// ---- VISUs/Estufa2.TcVIS
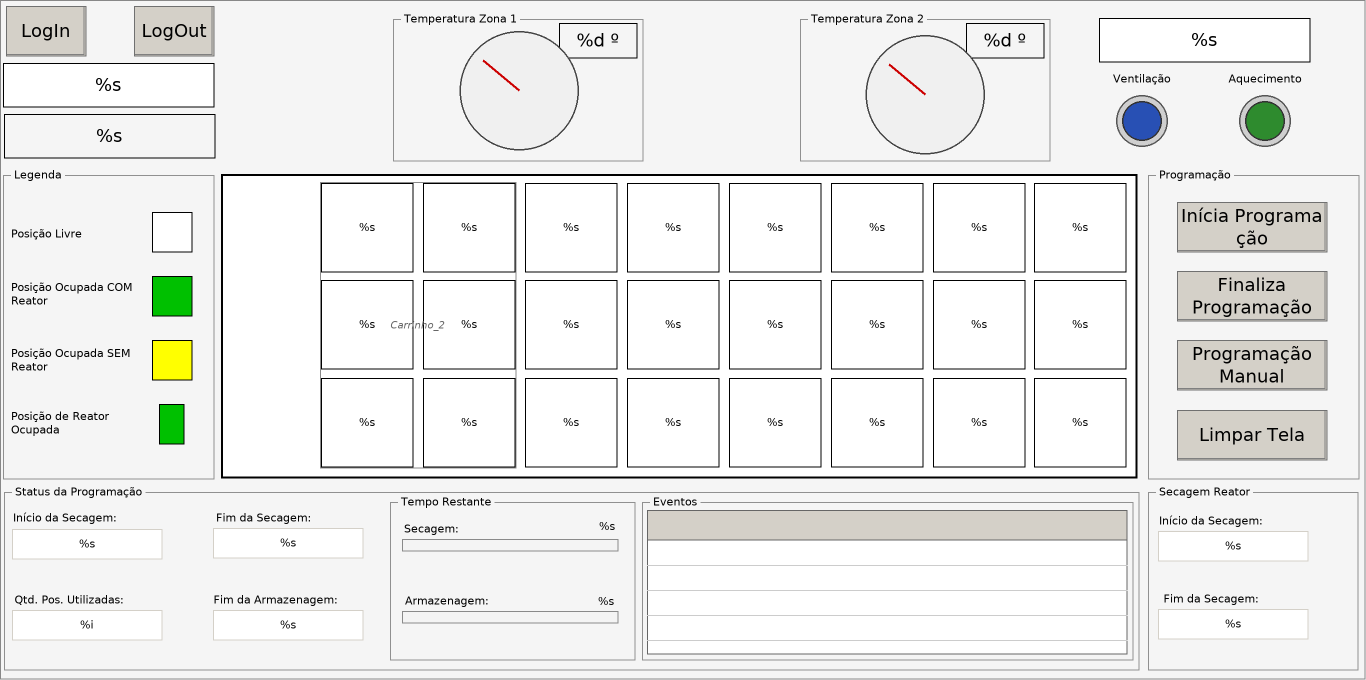
VISUALIZATION Estufa2  // 1366x680
    GroupBox (1148,484 210x186), "Secagem Reator", invisible if: GVL_P.bCarrinhoReator2
        Label (10,100 106x30), "Fim da Secagem:"
        Textfield (10,125 150x30), "%s", text variable: GVL_P.arrStatusEstufas[1].statusFimSecagem
    GroupBox (3,167 211x312), "Legenda"
        RoundedRectangle (149,173 40x40)
        RoundedRectangle (149,45 40x40)
        RoundedRectangle (156,237 25x40)
    GroupBox (800,11 250x150), "Temperatura Zona 2"
        Rectangle (166,12 78x35), "%d º", text variable: GVL.zona2atual_020
    GroupBox (393,11 250x150), "Temperatura Zona 1"
        Rectangle (166,12 78x35), "%d º", text variable: GVL.zona1atual_020
    GroupBox (4,484 1135x186), "Status da Programação"
        Label (209,19 101x30), "Fim da Secagem:"
        Label (209,101 125x30), "Fim da Armazenagem:"
        Label (8,101 114x30), "Qtd. Pos. Utilizadas:"
        GroupBox (638,10 491x166), "Eventos"
            Table (5,16 480x144), data array: GVL_P.arrLogEstufa20
                p3854506369: GVL_P.arrLogEstufa20[INDEX]
            InvisibleInput (7,16 431x142)
                OnMouseClick: OpenDialog Dialog=addComment, OpenModal=True, OpenCentered=True
        Label (8,19 106x30), "Início da Secagem:"
        Textfield (8,126 150x30), "%i", text variable: GVL.totalPos[1]
        Textfield (209,44 150x30), "%s", text variable: GVL_P.arrStatusEstufas[1].statusFimSecagem
        Textfield (209,126 150x30), "%s", text variable: GVL_P.arrStatusEstufas[1].statusFimArmazenagem
        GroupBox (386,10 245x166), "Tempo Restante"
            Progressbar (12,117 216x12), variable: MAIN.bardintArm20
            Rectangle (131,99 96x17), "%s", text variable: mid(str:=time_to_string(GVL.endArm20), LEN:= 20, POS:= 3)
            Progressbar (12,45 216x12), variable: MAIN.bardintSec20
        Label (398,30 59x30), "Secagem:"
    Rectangle (221,174 916x304)
    Meter180 (399,31 240x119), value: GVL.zona1atual_020, style: Meter-Meter180-Gray, scale format: %.1f, scale 20..160
        p518627256: ºC
    GroupBox (1148,167 211x312), "Programação"
        Button (29,35 150x50), "Inícia Programação", input disabled if: GVL_P.arrStatusEstufas[GVL.actEst].start
            OnMouseClick: OpenDialog Dialog=IniciaProg_2, OpenModal=True, OpenCentered=True
            OnMouseClick: execute { iniciaProgramacaoEstufa(); }
        Button (29,104 150x50), "Finaliza Programação"
            OnMouseClick: OpenDialog Dialog=FinalizaProg, Parameters={bReator: , iOFnumber: , iSrlNumber: }, OpenModal=True, OpenCentered=True
        Button (29,173 150x50), "Programação Manual", input disabled if: GVL_P.arrStatusEstufas[GVL.actEst].start
            OnMouseClick: OpenDialog Dialog=TimeCustom_2, OpenModal=True, OpenCentered=True
            OnMouseClick: execute { iniciaProgramacaoEstufa(); }
    Textfield (12,529 150x30), "%s", text variable: GVL_P.arrStatusEstufas[1].statusInicioSecagem
    Label (402,586 90x30), "Armazenagem:"
    Meter180 (805,35 240x119), value: GVL.zona2atual_020, style: Meter-Meter180-Gray, scale format: %.1f, scale 20..160
        p518627256: ºC
    RoundedRectangle (152,276 40x40)
    Label (8,278 132x32), "Posição Ocupada COM Reator"
    Label (8,344 128x32), "Posição Ocupada SEM Reator"
    Label (8,218 84x32), "Posição Livre"
    Label (8,407 128x32), "Posição de Reator Ocupada"
    Lamp1 (1112,91 60x60), variable: GVL.ventilacao_Ligada_020, style: Lamp-Lamp1-Blue
    Lamp1 (1235,91 60x60), variable: GVL.aquecimento_Ligado_020, style: Lamp-Lamp1-Green
    Label (1108,64 68x30), "Ventilação"
    Label (1227,64 76x30), "Aquecimento"
    Textfield (1158,531 150x30), "%s", text variable: GVL_P.arrStatusEstufas[1].inicioReator, invisible if: GVL_P.bCarrinhoReator2
    Label (1158,506 106x30), "Início da Secagem:", invisible if: GVL_P.bCarrinhoReator2
    Rectangle (1099,18 211x44), "%s", text variable: GVL_P.etapa_process[GVL.actEst]
    Rectangle (522,518 96x17), "%s", text variable: mid(str:=time_to_string(GVL.endSeca20), LEN:= 20, POS:= 3)
    Rectangle (1034,183 92x89), "%s", text variable: GVL_P.aPositionsE020[1].text, colour variable: GVL_P.aPositionsE020[1].color
        OnMouseUp: OpenDialog Dialog=ConfigPosicao_2, Parameters={bReator: , iOFnumber: , iSrlNumber: }, OpenModal=True, OpenCentered=True
        OnMouseUp: execute {
            gvl.actPos:=1;
            //selectPos021();
        }
    Rectangle (1034,280 92x89), "%s", text variable: GVL_P.aPositionsE020[2].text, colour variable: GVL_P.aPositionsE020[2].color
        OnMouseUp: OpenDialog Dialog=ConfigPosicao_2, Parameters={bReator: , iOFnumber: , iSrlNumber: }, OpenModal=True, OpenCentered=True
        OnMouseUp: execute {
            gvl.actPos:= 2;
            //selectPos021();
        }
    Rectangle (1034,378 92x89), "%s", text variable: GVL_P.aPositionsE020[3].text, colour variable: GVL_P.aPositionsE020[3].color
        OnMouseUp: OpenDialog Dialog=ConfigPosicao_2, Parameters={bReator: , iOFnumber: , iSrlNumber: }, OpenModal=True, OpenCentered=True
        OnMouseUp: execute {
            gvl.actPos:= 3;
            //selectPos021();
        }
    Rectangle (933,183 92x89), "%s", text variable: GVL_P.aPositionsE020[4].text, colour variable: GVL_P.aPositionsE020[4].color
        OnMouseUp: OpenDialog Dialog=ConfigPosicao_2, Parameters={bReator: , iOFnumber: , iSrlNumber: }, OpenModal=True, OpenCentered=True
        OnMouseUp: execute {
            gvl.actPos:= 4;
            //selectPos021();
        }
    Rectangle (933,280 92x89), "%s", text variable: GVL_P.aPositionsE020[5].text, colour variable: GVL_p.aPositionsE020[5].color
        OnMouseUp: OpenDialog Dialog=ConfigPosicao_2, Parameters={bReator: , iOFnumber: , iSrlNumber: }, OpenModal=True, OpenCentered=True
        OnMouseUp: execute {
            gvl.actPos:= 5;
            //selectPos021();
        }
    Rectangle (933,378 92x89), "%s", text variable: GVL_P.aPositionsE020[6].text, colour variable: GVL_P.aPositionsE020[6].color
        OnMouseUp: OpenDialog Dialog=ConfigPosicao_2, Parameters={bReator: , iOFnumber: , iSrlNumber: }, OpenModal=True, OpenCentered=True
        OnMouseUp: execute {
            gvl.actPos:= 6;
            //selectPos021();
        }
    Rectangle (831,183 92x89), "%s", text variable: GVL_P.aPositionsE020[7].text, colour variable: GVL_P.aPositionsE020[7].color
        OnMouseUp: OpenDialog Dialog=ConfigPosicao_2, Parameters={bReator: , iOFnumber: , iSrlNumber: }, OpenModal=True, OpenCentered=True
        OnMouseUp: execute {
            gvl.actPos:= 7;
            //selectPos021();
        }
    Rectangle (831,280 92x89), "%s", text variable: GVL_P.aPositionsE020[8].text, colour variable: GVL_P.aPositionsE020[8].color
        OnMouseUp: OpenDialog Dialog=ConfigPosicao_2, Parameters={bReator: , iOFnumber: , iSrlNumber: }, OpenModal=True, OpenCentered=True
        OnMouseUp: execute {
            gvl.actPos:= 8;
            //selectPos021();
        }
    Rectangle (831,378 92x89), "%s", text variable: GVL_P.aPositionsE020[9].text, colour variable: GVL_P.aPositionsE020[9].color
        OnMouseUp: OpenDialog Dialog=ConfigPosicao_2, Parameters={bReator: , iOFnumber: , iSrlNumber: }, OpenModal=True, OpenCentered=True
        OnMouseUp: execute {
            gvl.actPos:= 9;
            //selectPos021();
        }
    Rectangle (729,183 92x89), "%s", text variable: GVL_P.aPositionsE020[10].text, colour variable: GVL_P.aPositionsE020[10].color
        OnMouseUp: OpenDialog Dialog=ConfigPosicao_2, Parameters={bReator: , iOFnumber: , iSrlNumber: }, OpenModal=True, OpenCentered=True
        OnMouseUp: execute {
            gvl.actPos:= 10;
            //selectPos021();
        }
    Rectangle (729,280 92x89), "%s", text variable: GVL_P.aPositionsE020[11].text, colour variable: GVL_P.aPositionsE020[11].color
        OnMouseUp: OpenDialog Dialog=ConfigPosicao_2, Parameters={bReator: , iOFnumber: , iSrlNumber: }, OpenModal=True, OpenCentered=True
        OnMouseUp: execute {
            gvl.actPos:= 11;
            //selectPos021();
        }
    Rectangle (729,378 92x89), "%s", text variable: GVL_P.aPositionsE020[12].text, colour variable: GVL_P.aPositionsE020[12].color
        OnMouseUp: OpenDialog Dialog=ConfigPosicao_2, Parameters={bReator: , iOFnumber: , iSrlNumber: }, OpenModal=True, OpenCentered=True
        OnMouseUp: execute {
            gvl.actPos:= 12;
            //selectPos021();
        }
    Rectangle (627,183 92x89), "%s", text variable: GVL_P.aPositionsE020[13].text, colour variable: GVL_P.aPositionsE020[13].color
        OnMouseUp: OpenDialog Dialog=ConfigPosicao_2, Parameters={bReator: , iOFnumber: , iSrlNumber: }, OpenModal=True, OpenCentered=True
        OnMouseUp: execute {
            gvl.actPos:= 13;
            //selectPos021();
        }
    Rectangle (627,280 92x89), "%s", text variable: GVL_P.aPositionsE020[14].text, colour variable: GVL_P.aPositionsE020[14].color
        OnMouseUp: OpenDialog Dialog=ConfigPosicao_2, Parameters={bReator: , iOFnumber: , iSrlNumber: }, OpenModal=True, OpenCentered=True
        OnMouseUp: execute {
            gvl.actPos:= 14;
            //selectPos021();
        }
    Rectangle (627,378 92x89), "%s", text variable: GVL_P.aPositionsE020[15].text, colour variable: GVL_P.aPositionsE020[15].color
        OnMouseUp: OpenDialog Dialog=ConfigPosicao_2, Parameters={bReator: , iOFnumber: , iSrlNumber: }, OpenModal=True, OpenCentered=True
        OnMouseUp: execute {
            gvl.actPos:= 15;
            //selectPos021();
        }
    Rectangle (525,183 92x89), "%s", text variable: GVL_P.aPositionsE020[16].text, colour variable: GVL_P.aPositionsE020[16].color
        OnMouseUp: OpenDialog Dialog=ConfigPosicao_2, Parameters={bReator: , iOFnumber: , iSrlNumber: }, OpenModal=True, OpenCentered=True
        OnMouseUp: execute {
            gvl.actPos:= 16;
            //selectPos021();
        }
    Rectangle (525,280 92x89), "%s", text variable: GVL_P.aPositionsE020[17].text, colour variable: GVL_P.aPositionsE020[17].color
        OnMouseUp: OpenDialog Dialog=ConfigPosicao_2, Parameters={bReator: , iOFnumber: , iSrlNumber: }, OpenModal=True, OpenCentered=True
        OnMouseUp: execute {
            gvl.actPos:= 17;
            //selectPos021();
        }
    Rectangle (525,378 92x89), "%s", text variable: GVL_P.aPositionsE020[18].text, colour variable: GVL_P.aPositionsE020[18].color
        OnMouseUp: OpenDialog Dialog=ConfigPosicao_2, Parameters={bReator: , iOFnumber: , iSrlNumber: }, OpenModal=True, OpenCentered=True
        OnMouseUp: execute {
            gvl.actPos:= 18;
            //selectPos021();
        }
    Rectangle (423,183 92x89), "%s", text variable: GVL_P.aPositionsE020[19].text, colour variable: GVL_P.aPositionsE020[19].color
        OnMouseUp: OpenDialog Dialog=ConfigPosicao_2, Parameters={bReator: , iOFnumber: , iSrlNumber: }, OpenModal=True, OpenCentered=True
        OnMouseUp: execute {
            gvl.actPos:= 19;
            //selectPos021();
        }
    Rectangle (423,280 92x89), "%s", text variable: GVL_P.aPositionsE020[20].text, colour variable: GVL_P.aPositionsE020[20].color
        OnMouseUp: OpenDialog Dialog=ConfigPosicao_2, Parameters={bReator: , iOFnumber: , iSrlNumber: }, OpenModal=True, OpenCentered=True
        OnMouseUp: execute {
            gvl.actPos:= 20;
            //selectPos021();
        }
    Rectangle (423,378 92x89), "%s", text variable: GVL_P.aPositionsE020[21].text, colour variable: GVL_P.aPositionsE020[21].color
        OnMouseUp: OpenDialog Dialog=ConfigPosicao_2, Parameters={bReator: , iOFnumber: , iSrlNumber: }, OpenModal=True, OpenCentered=True
        OnMouseUp: execute {
            gvl.actPos:= 21;
            //selectPos021();
        }
    Rectangle (321,183 92x89), "%s", text variable: GVL_P.aPositionsE020[22].text, colour variable: GVL_P.aPositionsE020[22].color
        OnMouseUp: OpenDialog Dialog=ConfigPosicao_2, Parameters={bReator: , iOFnumber: , iSrlNumber: }, OpenModal=True, OpenCentered=True
        OnMouseUp: execute {
            gvl.actPos:= 22;
            //selectPos021();
        }
    Rectangle (321,280 92x89), "%s", text variable: GVL_P.aPositionsE020[23].text, colour variable: GVL_P.aPositionsE020[23].color
        OnMouseUp: OpenDialog Dialog=ConfigPosicao_2, Parameters={bReator: , iOFnumber: , iSrlNumber: }, OpenModal=True, OpenCentered=True
        OnMouseUp: execute {
            gvl.actPos:= 23;
            //selectPos021();
        }
    Rectangle (321,378 92x89), "%s", text variable: GVL_P.aPositionsE020[24].text, colour variable: GVL_P.aPositionsE020[24].color
        OnMouseUp: OpenDialog Dialog=ConfigPosicao_2, Parameters={bReator: , iOFnumber: , iSrlNumber: }, OpenModal=True, OpenCentered=True
        OnMouseUp: execute {
            gvl.actPos:= 24;
            //selectPos021();
        }
    Frame (320,182 196x286), invisible if: GVL_P.bCarrinhoReator2
        shows Carrinho_2()
    Button (1177,410 150x50), "Limpar Tela"
        OnMouseClick: execute {
            FOR gvl.i:=1 TO 24 BY 1 DO
            gvl_p.aPositionsE020[gvl.i].numOF:='';
            gvl_p.aPositionsE020[gvl.i].lote:='';
            gvl_p.aPositionsE020[gvl.i].class:=0;
            gvl_p.aPositionsE020[gvl.i].pot:=0;
            gvl_p.aPositionsE020[gvl.i].cor:=0;
            gvl_p.aPositionsE020[gvl.i].text:='';
            gvl_p.aPositionsE020[gvl.i].reator:=true;
            END_FOR
            FOR gvl.i:=1 TO 18 BY 1 DO
            gvl_p.corPosReator2[gvl.i].cor:=0;
            END_FOR
            gravarConfigPosicao.bReator[1]:= FALSE;
            ///// GERADOR DE LOG -------------------------------------------------------------
            gvl.envialog:= 'Todas as posições foram limpas. ESTUFA 20';
            gvl.logRegister20:= gvl.envialog;
            gvl.sCmdInsertLog:= 'INSERT INTO [dbo].[LogGeneral] ([HistoricalTime],[Description])VALUES($'$',$'$')';
            gvl.sCmdInsertLog:= insert(gvl.sCmdInsertLog,gvl.logRegister20,74);
            gvl.sCmdInsertLog:= insert(gvl.sCmdInsertLog,gvl.sSystemDateTime,71);
            gvl.bInsertLog:= TRUE;
        }
    Rectangle (3,63 211x44), "%s", text variable: MAIN.sDB_Operador
    Rectangle (4,114 211x44), "%s", text variable: GVL.sSystemTime
    Button (6,6 80x50), "LogIn"
        OnMouseClick: VisuUserMgmt Type=Login
    Button (134,6 80x50), "LogOut"
        OnMouseClick: VisuUserMgmt Type=Logout
END_VISUALIZATION

// ---- VISUs/Estufa3.TcVIS
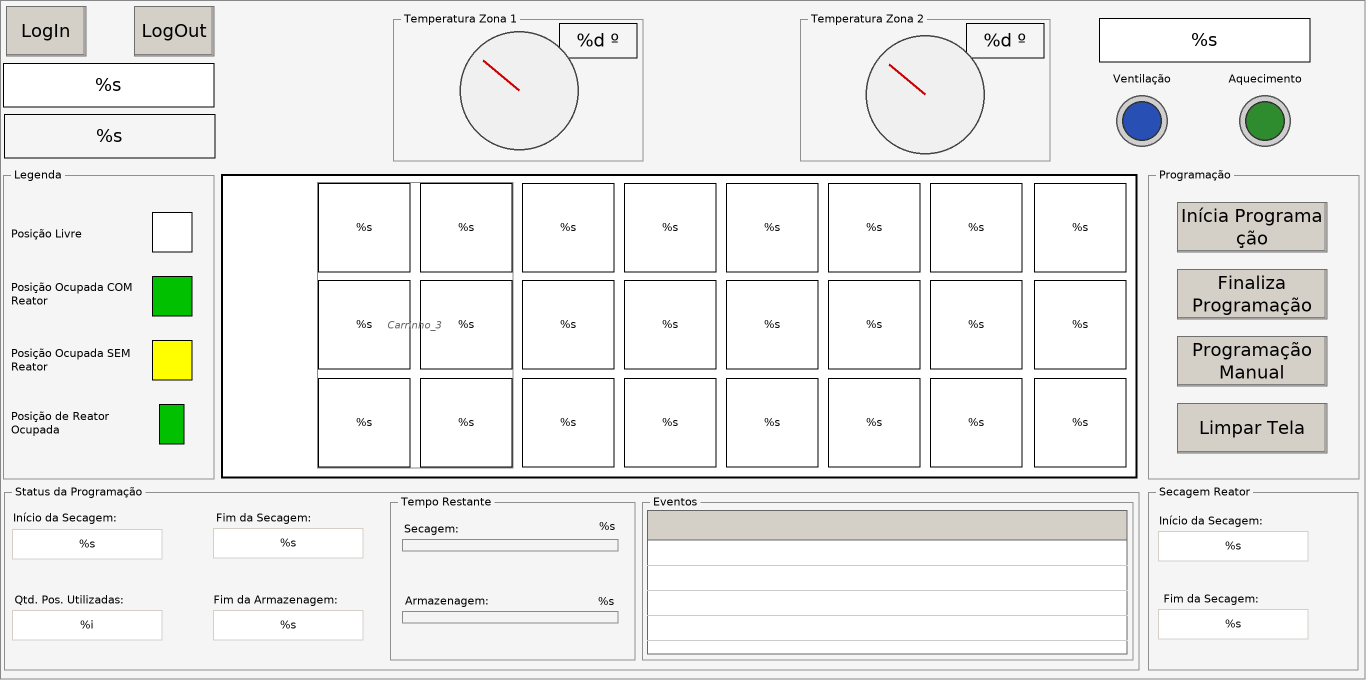
VISUALIZATION Estufa3  // 1366x680
    GroupBox (1148,484 210x186), "Secagem Reator", invisible if: GVL_P.bCarrinhoReator3
        Label (10,100 106x30), "Fim da Secagem:"
        Textfield (10,125 150x30), "%s", text variable: GVL_P.arrStatusEstufas[2].statusFimSecagem
    GroupBox (3,167 211x312), "Legenda"
        RoundedRectangle (149,173 40x40)
        RoundedRectangle (149,45 40x40)
        RoundedRectangle (156,237 25x40)
    GroupBox (800,11 250x150), "Temperatura Zona 2"
        Rectangle (166,12 78x35), "%d º", text variable: GVL.zona2atual_021
    GroupBox (393,11 250x150), "Temperatura Zona 1"
        Rectangle (166,12 78x35), "%d º", text variable: GVL.zona1atual_021
    GroupBox (4,484 1135x186), "Status da Programação"
        Label (209,19 101x30), "Fim da Secagem:"
        Label (209,101 125x30), "Fim da Armazenagem:"
        Label (8,101 114x30), "Qtd. Pos. Utilizadas:"
        GroupBox (638,10 491x166), "Eventos"
            Table (5,16 480x144), data array: GVL_P.arrLogEstufa21
                p3854506369: GVL_P.arrLogEstufa21[INDEX]
            InvisibleInput (7,16 431x142)
                OnMouseClick: OpenDialog Dialog=addComment, OpenModal=True, OpenCentered=True
        Label (8,19 106x30), "Início da Secagem:"
        Textfield (8,126 150x30), "%i", text variable: GVL.totalPos[2]
        Textfield (209,44 150x30), "%s", text variable: GVL_P.arrStatusEstufas[2].statusFimSecagem
        Textfield (209,126 150x30), "%s", text variable: GVL_P.arrStatusEstufas[2].statusFimArmazenagem
        GroupBox (386,10 245x166), "Tempo Restante"
            Progressbar (12,117 216x12), variable: MAIN.bardintArm21
            Rectangle (131,99 96x17), "%s", text variable: mid(str:=time_to_string(GVL.endArm21), LEN:= 20, POS:= 3)
            Progressbar (12,45 216x12), variable: MAIN.bardintSec21
        Label (398,30 59x30), "Secagem:"
    Rectangle (221,174 916x304)
    Rectangle (1034,183 92x89), "%s", text variable: GVL_P.aPositionsE021[1].text, colour variable: GVL_P.aPositionsE021[1].color
        OnMouseUp: OpenDialog Dialog=ConfigPosicao_3, Parameters={bReator: , iOFnumber: , iSrlNumber: }, OpenModal=True, OpenCentered=True
        OnMouseUp: execute {
            gvl.actPos:=1;
            //selectPos021();
        }
    Rectangle (1034,280 92x89), "%s", text variable: GVL_P.aPositionsE021[2].text, colour variable: GVL_P.aPositionsE021[2].color
        OnMouseUp: OpenDialog Dialog=ConfigPosicao_3, Parameters={bReator: , iOFnumber: , iSrlNumber: }, OpenModal=True, OpenCentered=True
        OnMouseUp: execute {
            gvl.actPos:= 2;
            //selectPos021();
        }
    Rectangle (1034,378 92x89), "%s", text variable: GVL_P.aPositionsE021[3].text, colour variable: GVL_P.aPositionsE021[3].color
        OnMouseUp: OpenDialog Dialog=ConfigPosicao_3, Parameters={bReator: , iOFnumber: , iSrlNumber: }, OpenModal=True, OpenCentered=True
        OnMouseUp: execute {
            gvl.actPos:= 3;
            //selectPos021();
        }
    Rectangle (930,183 92x89), "%s", text variable: GVL_P.aPositionsE021[4].text, colour variable: GVL_P.aPositionsE021[4].color
        OnMouseUp: OpenDialog Dialog=ConfigPosicao_3, Parameters={bReator: , iOFnumber: , iSrlNumber: }, OpenModal=True, OpenCentered=True
        OnMouseUp: execute {
            gvl.actPos:= 4;
            //selectPos021();
        }
    Rectangle (930,280 92x89), "%s", text variable: GVL_P.aPositionsE021[5].text, colour variable: GVL_p.aPositionsE021[5].color
        OnMouseUp: OpenDialog Dialog=ConfigPosicao_3, Parameters={bReator: , iOFnumber: , iSrlNumber: }, OpenModal=True, OpenCentered=True
        OnMouseUp: execute {
            gvl.actPos:= 5;
            //selectPos021();
        }
    Rectangle (930,378 92x89), "%s", text variable: GVL_P.aPositionsE021[6].text, colour variable: GVL_P.aPositionsE021[6].color
        OnMouseUp: OpenDialog Dialog=ConfigPosicao_3, Parameters={bReator: , iOFnumber: , iSrlNumber: }, OpenModal=True, OpenCentered=True
        OnMouseUp: execute {
            gvl.actPos:= 6;
            //selectPos021();
        }
    Rectangle (828,183 92x89), "%s", text variable: GVL_P.aPositionsE021[7].text, colour variable: GVL_P.aPositionsE021[7].color
        OnMouseUp: OpenDialog Dialog=ConfigPosicao_3, Parameters={bReator: , iOFnumber: , iSrlNumber: }, OpenModal=True, OpenCentered=True
        OnMouseUp: execute {
            gvl.actPos:= 7;
            //selectPos021();
        }
    Rectangle (828,280 92x89), "%s", text variable: GVL_P.aPositionsE021[8].text, colour variable: GVL_P.aPositionsE021[8].color
        OnMouseUp: OpenDialog Dialog=ConfigPosicao_3, Parameters={bReator: , iOFnumber: , iSrlNumber: }, OpenModal=True, OpenCentered=True
        OnMouseUp: execute {
            gvl.actPos:= 8;
            //selectPos021();
        }
    Rectangle (828,378 92x89), "%s", text variable: GVL_P.aPositionsE021[9].text, colour variable: GVL_P.aPositionsE021[9].color
        OnMouseUp: OpenDialog Dialog=ConfigPosicao_3, Parameters={bReator: , iOFnumber: , iSrlNumber: }, OpenModal=True, OpenCentered=True
        OnMouseUp: execute {
            gvl.actPos:= 9;
            //selectPos021();
        }
    Rectangle (726,183 92x89), "%s", text variable: GVL_P.aPositionsE021[10].text, colour variable: GVL_P.aPositionsE021[10].color
        OnMouseUp: OpenDialog Dialog=ConfigPosicao_3, Parameters={bReator: , iOFnumber: , iSrlNumber: }, OpenModal=True, OpenCentered=True
        OnMouseUp: execute {
            gvl.actPos:= 10;
            //selectPos021();
        }
    Rectangle (726,280 92x89), "%s", text variable: GVL_P.aPositionsE021[11].text, colour variable: GVL_P.aPositionsE021[11].color
        OnMouseUp: OpenDialog Dialog=ConfigPosicao_3, Parameters={bReator: , iOFnumber: , iSrlNumber: }, OpenModal=True, OpenCentered=True
        OnMouseUp: execute {
            gvl.actPos:= 11;
            //selectPos021();
        }
    Rectangle (726,378 92x89), "%s", text variable: GVL_P.aPositionsE021[12].text, colour variable: GVL_P.aPositionsE021[12].color
        OnMouseUp: OpenDialog Dialog=ConfigPosicao_3, Parameters={bReator: , iOFnumber: , iSrlNumber: }, OpenModal=True, OpenCentered=True
        OnMouseUp: execute {
            gvl.actPos:= 12;
            //selectPos021();
        }
    Rectangle (624,183 92x89), "%s", text variable: GVL_P.aPositionsE021[13].text, colour variable: GVL_P.aPositionsE021[13].color
        OnMouseUp: OpenDialog Dialog=ConfigPosicao_3, Parameters={bReator: , iOFnumber: , iSrlNumber: }, OpenModal=True, OpenCentered=True
        OnMouseUp: execute {
            gvl.actPos:= 13;
            //selectPos021();
        }
    Rectangle (624,280 92x89), "%s", text variable: GVL_P.aPositionsE021[14].text, colour variable: GVL_P.aPositionsE021[14].color
        OnMouseUp: OpenDialog Dialog=ConfigPosicao_3, Parameters={bReator: , iOFnumber: , iSrlNumber: }, OpenModal=True, OpenCentered=True
        OnMouseUp: execute {
            gvl.actPos:= 14;
            //selectPos021();
        }
    Rectangle (624,378 92x89), "%s", text variable: GVL_P.aPositionsE021[15].text, colour variable: GVL_P.aPositionsE021[15].color
        OnMouseUp: OpenDialog Dialog=ConfigPosicao_3, Parameters={bReator: , iOFnumber: , iSrlNumber: }, OpenModal=True, OpenCentered=True
        OnMouseUp: execute {
            gvl.actPos:= 15;
            //selectPos021();
        }
    Rectangle (522,183 92x89), "%s", text variable: GVL_P.aPositionsE021[16].text, colour variable: GVL_P.aPositionsE021[16].color
        OnMouseUp: OpenDialog Dialog=ConfigPosicao_3, Parameters={bReator: , iOFnumber: , iSrlNumber: }, OpenModal=True, OpenCentered=True
        OnMouseUp: execute {
            gvl.actPos:= 16;
            //selectPos021();
        }
    Rectangle (522,280 92x89), "%s", text variable: GVL_P.aPositionsE021[17].text, colour variable: GVL_P.aPositionsE021[17].color
        OnMouseUp: OpenDialog Dialog=ConfigPosicao_3, Parameters={bReator: , iOFnumber: , iSrlNumber: }, OpenModal=True, OpenCentered=True
        OnMouseUp: execute {
            gvl.actPos:= 17;
            //selectPos021();
        }
    Rectangle (522,378 92x89), "%s", text variable: GVL_P.aPositionsE021[18].text, colour variable: GVL_P.aPositionsE021[18].color
        OnMouseUp: OpenDialog Dialog=ConfigPosicao_3, Parameters={bReator: , iOFnumber: , iSrlNumber: }, OpenModal=True, OpenCentered=True
        OnMouseUp: execute {
            gvl.actPos:= 18;
            //selectPos021();
        }
    Rectangle (420,183 92x89), "%s", text variable: GVL_P.aPositionsE021[19].text, colour variable: GVL_P.aPositionsE021[19].color
        OnMouseUp: OpenDialog Dialog=ConfigPosicao_3, Parameters={bReator: , iOFnumber: , iSrlNumber: }, OpenModal=True, OpenCentered=True
        OnMouseUp: execute {
            gvl.actPos:= 19;
            //selectPos021();
        }
    Rectangle (420,280 92x89), "%s", text variable: GVL_P.aPositionsE021[20].text, colour variable: GVL_P.aPositionsE021[20].color
        OnMouseUp: OpenDialog Dialog=ConfigPosicao_3, Parameters={bReator: , iOFnumber: , iSrlNumber: }, OpenModal=True, OpenCentered=True
        OnMouseUp: execute {
            gvl.actPos:= 20;
            //selectPos021();
        }
    Rectangle (420,378 92x89), "%s", text variable: GVL_P.aPositionsE021[21].text, colour variable: GVL_P.aPositionsE021[21].color
        OnMouseUp: OpenDialog Dialog=ConfigPosicao_3, Parameters={bReator: , iOFnumber: , iSrlNumber: }, OpenModal=True, OpenCentered=True
        OnMouseUp: execute {
            gvl.actPos:= 21;
            //selectPos021();
        }
    Rectangle (318,183 92x89), "%s", text variable: GVL_P.aPositionsE021[22].text, colour variable: GVL_P.aPositionsE021[22].color
        OnMouseUp: OpenDialog Dialog=ConfigPosicao_3, Parameters={bReator: , iOFnumber: , iSrlNumber: }, OpenModal=True, OpenCentered=True
        OnMouseUp: execute {
            gvl.actPos:= 22;
            //selectPos021();
        }
    Rectangle (318,280 92x89), "%s", text variable: GVL_P.aPositionsE021[23].text, colour variable: GVL_P.aPositionsE021[23].color
        OnMouseUp: OpenDialog Dialog=ConfigPosicao_3, Parameters={bReator: , iOFnumber: , iSrlNumber: }, OpenModal=True, OpenCentered=True
        OnMouseUp: execute {
            gvl.actPos:= 23;
            //selectPos021();
        }
    Rectangle (318,378 92x89), "%s", text variable: GVL_P.aPositionsE021[24].text, colour variable: GVL_P.aPositionsE021[24].color
        OnMouseUp: OpenDialog Dialog=ConfigPosicao_3, Parameters={bReator: , iOFnumber: , iSrlNumber: }, OpenModal=True, OpenCentered=True
        OnMouseUp: execute {
            gvl.actPos:= 24;
            //selectPos021();
        }
    Meter180 (399,31 240x119), value: GVL.zona1atual_021, style: Meter-Meter180-Gray, scale format: %.1f, scale 20..160
        p518627256: ºC
    GroupBox (1148,167 211x312), "Programação"
        Button (29,35 150x50), "Inícia Programação", input disabled if: GVL_P.arrStatusEstufas[GVL.actEst].start
            OnMouseClick: OpenDialog Dialog=IniciaProg_3, OpenModal=True, OpenCentered=True
            OnMouseClick: execute { iniciaProgramacaoEstufa(); }
        Button (29,102 150x50), "Finaliza Programação"
            OnMouseClick: OpenDialog Dialog=FinalizaProg, Parameters={bReator: , iOFnumber: , iSrlNumber: }, OpenModal=True, OpenCentered=True
        Button (29,169 150x50), "Programação Manual", input disabled if: GVL_P.arrStatusEstufas[GVL.actEst].start
            OnMouseClick: OpenDialog Dialog=TimeCustom_3, OpenModal=True, OpenCentered=True
            OnMouseClick: execute { iniciaProgramacaoEstufa(); }
    Textfield (12,529 150x30), "%s", text variable: GVL_P.arrStatusEstufas[2].statusInicioSecagem
    Label (402,586 90x30), "Armazenagem:"
    Meter180 (805,35 240x119), value: GVL.zona2atual_021, style: Meter-Meter180-Gray, scale format: %.1f, scale 20..160
        p518627256: ºC
    RoundedRectangle (152,276 40x40)
    Label (8,278 132x32), "Posição Ocupada COM Reator"
    Label (8,344 128x32), "Posição Ocupada SEM Reator"
    Label (8,218 84x32), "Posição Livre"
    Label (8,407 128x32), "Posição de Reator Ocupada"
    Frame (317,182 196x286), invisible if: GVL_P.bCarrinhoReator3
        shows Carrinho_3()
    Lamp1 (1112,91 60x60), variable: GVL.ventilacao_Ligada_021, style: Lamp-Lamp1-Blue
    Lamp1 (1235,91 60x60), variable: GVL.aquecimento_Ligado_021, style: Lamp-Lamp1-Green
    Label (1108,64 68x30), "Ventilação"
    Label (1227,64 76x30), "Aquecimento"
    Textfield (1158,531 150x30), "%s", text variable: GVL_P.arrStatusEstufas[2].inicioReator, invisible if: GVL_P.bCarrinhoReator3
    Label (1158,506 106x30), "Início da Secagem:", invisible if: GVL_P.bCarrinhoReator3
    Rectangle (1099,18 211x44), "%s", text variable: GVL_P.etapa_process[GVL.actEst]
    Rectangle (522,518 96x17), "%s", text variable: mid(str:=time_to_string(GVL.endSeca21), LEN:= 20, POS:= 3)
    Button (1177,403 150x50), "Limpar Tela"
        OnMouseClick: execute {
            FOR gvl.i:=1 TO 24 BY 1 DO
            gvl_p.aPositionsE021[gvl.i].numOF:='';
            gvl_p.aPositionsE021[gvl.i].lote:='';
            gvl_p.aPositionsE021[gvl.i].class:=0;
            gvl_p.aPositionsE021[gvl.i].pot:=0;
            gvl_p.aPositionsE021[gvl.i].cor:=0;
            gvl_p.aPositionsE021[gvl.i].text:='';
            gvl_p.aPositionsE021[gvl.i].reator:=true;
            END_FOR
            FOR gvl.i:=1 TO 18 BY 1 DO
            gvl_p.corPosReator3[gvl.i].cor:=0;
            END_FOR
            gravarConfigPosicao.bReator[2]:= FALSE;
            ///// GERADOR DE LOG -------------------------------------------------------------
            gvl.envialog:= 'Todas as posições foram limpas. ESTUFA 21';
            gvl.logRegister21:= gvl.envialog;
            gvl.sCmdInsertLog:= 'INSERT INTO [dbo].[LogGeneral] ([HistoricalTime],[Description])VALUES($'$',$'$')';
            gvl.sCmdInsertLog:= insert(gvl.sCmdInsertLog,gvl.logRegister21,74);
            gvl.sCmdInsertLog:= insert(gvl.sCmdInsertLog,gvl.sSystemDateTime,71);
            gvl.bInsertLog:= TRUE;
        }
    Rectangle (3,63 211x44), "%s", text variable: MAIN.sDB_Operador
    Rectangle (4,114 211x44), "%s", text variable: GVL.sSystemTime
    Button (6,6 80x50), "LogIn"
        OnMouseClick: VisuUserMgmt Type=Login
    Button (134,6 80x50), "LogOut"
        OnMouseClick: VisuUserMgmt Type=Logout
END_VISUALIZATION

// ---- VISUs/FinalizaProg.TcVIS
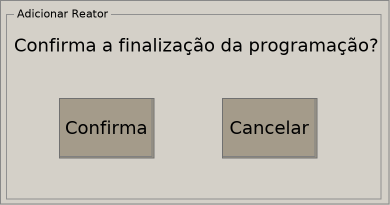
VISUALIZATION FinalizaProg  // 390x205
VAR_IN_OUT
	bReator: BOOL;
	iOFnumber: INT;
	iSrlNumber: INT;
	
	
	
END_VAR
    GroupBox (6,6 375x193), "Adicionar Reator"
        Button (53,92 95x60), "Confirma"
            OnMouseClick: CloseDialog Dialog=FinalizaProg, Result=OK, NumpadKeypadSet=True
            OnMouseClick: execute {
                IF gvl.actEst = 0 THEN
                	Rotina019.status:= 45;
                	Rotina019_Manual.status:= 45;
                ELSIF gvl.actEst = 1 THEN
                	Rotina020.status:= 45;
                	Rotina020_Manual.status:=45;
                ELSIF gvl.actEst = 2 THEN
                	Rotina021.status:= 45;
                	Rotina021_Manual.status:= 45;
                END_IF
            }
        Button (216,92 95x60), "Cancelar"
            OnMouseClick: CloseDialog Dialog=FinalizaProg, Result=Cancel, NumpadKeypadSet=True
        Label (5,27 381x63), "Confirma a finalização da programação?"
END_VISUALIZATION

// ---- VISUs/Grafico_3.TcVIS
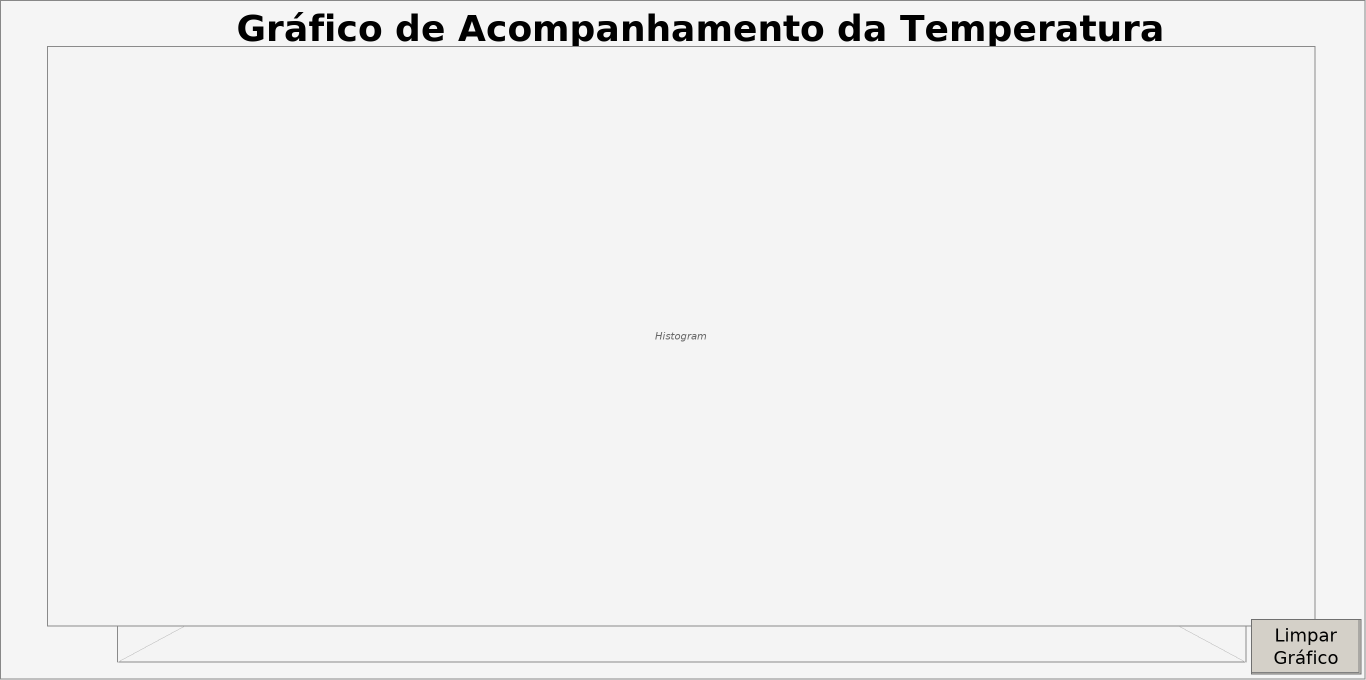
VISUALIZATION Grafico_3  // 1366x680
    Image (117,53 1129x609), image: ImagePool.Screenshot_3
    Histogram (47,46 1268x580), scale format: %.1f, scale 0..150
        p1518820177: GVL_P.arrTempVisu021
        p102497268: GVL_P.arrTempVisu021
        p788070771: ARRAY [1..720] OF REAL
    Label (262,7 877x43), "Gráfico de Acompanhamento da Temperatura"
    Histogram (47,46 1268x580), scale format: %.1f, scale 0..150
        p1518820177: GVL_P.arrTemp021
        p102497268: GVL_P.arrTemp021
        p788070771: ARRAY [1..720] OF REAL
    Button (1251,619 110x55), "Limpar Gráfico"
        OnMouseClick: execute {
            FOR gvl.i:=0 TO 720 BY 1 DO
            	gvl_p.arrTemp021[gvl.i]:= 0;
            	gvl_p.arrTempVisu021[gvl.i]:= 0;
            	END_FOR
        }
END_VISUALIZATION

// ---- VISUs/Grafico_2.TcVIS
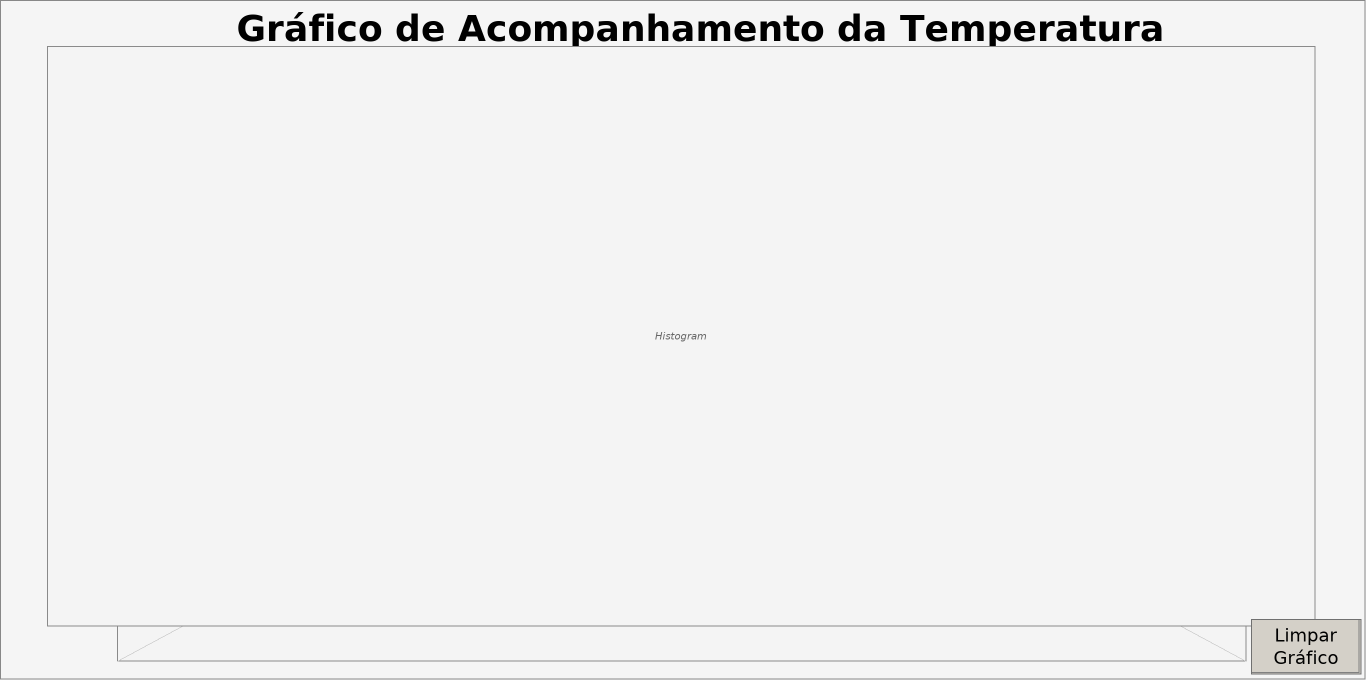
VISUALIZATION Grafico_2  // 1366x680
    Image (117,52 1129x609), image: ImagePool.Screenshot_3
    Histogram (47,46 1268x580), scale format: %.1f, scale 0..150
        p1518820177: GVL_P.arrTempVisu020
        p102497268: GVL_P.arrTempVisu020
        p788070771: ARRAY [1..720] OF REAL
    Label (262,7 877x43), "Gráfico de Acompanhamento da Temperatura"
    Histogram (47,46 1268x580), scale format: %.1f, scale 0..150
        p1518820177: GVL_P.arrTemp020
        p102497268: GVL_P.arrTemp020
        p788070771: ARRAY [1..720] OF REAL
    Button (1251,619 110x55), "Limpar Gráfico"
        OnMouseClick: execute {
            FOR gvl.i:=0 TO 720 BY 1 DO
            	gvl_p.arrTemp020[gvl.i]:= 0;
            	gvl_p.arrTempVisu020[gvl.i]:= 0;
            	END_FOR
        }
END_VISUALIZATION

// ---- VISUs/Historical.TcVIS
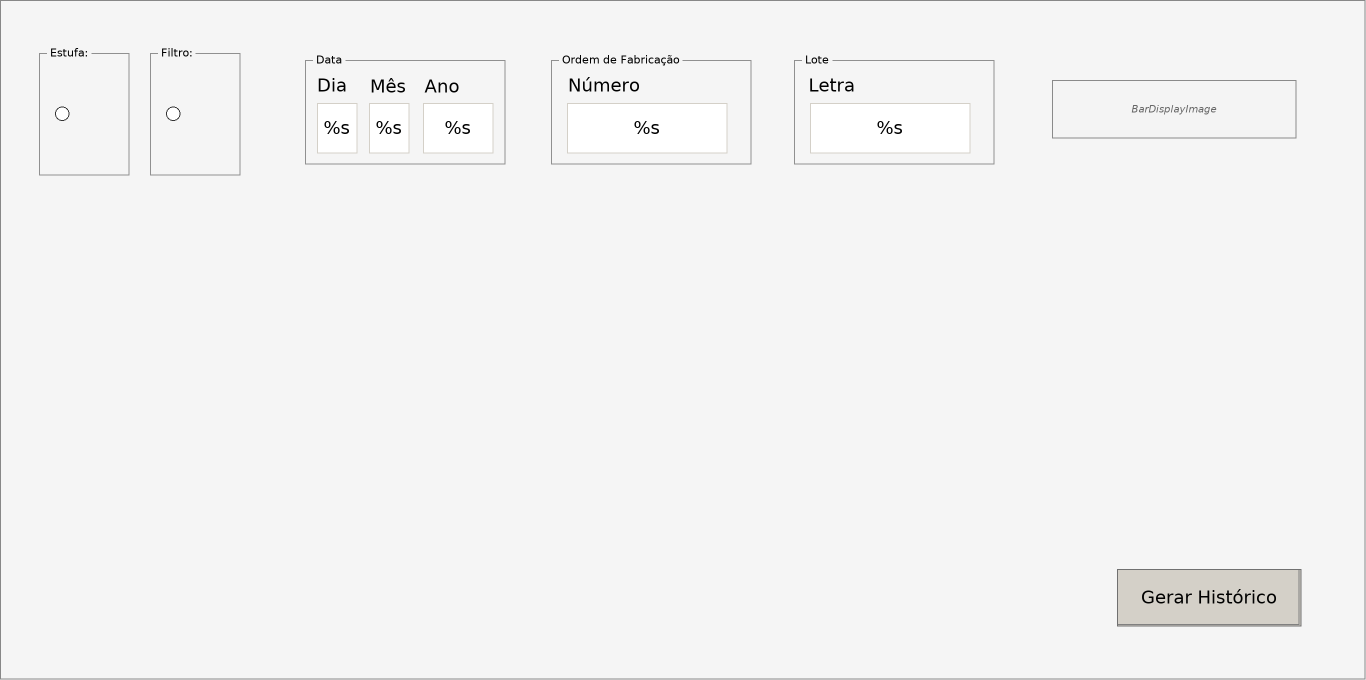
VISUALIZATION Historical  // 1366x680
    GroupBox (39,45 90x130), "Estufa:"
        RadioButton (14,24 65x89), variable: GVL.radioEstufa
            Areas[0]: Text=019
            Areas[1]: Text=020
            Areas[2]: Text=021
    Textfield (317,103 40x50), "%s", text variable: GVL.arrCVSfilter[GVL.radioEstufa].dia, input disabled if: GVL.radioData
        OnMouseClick: write the text variable via VisuDialogs.Numpad
    GroupBox (150,45 90x130), "Filtro:"
        RadioButton (14,24 65x89), variable: GVL.radioFiltro
            Areas[0]: Text=Data
            Areas[2]: Text=Lote
    BarDisplayImage (1052,80 244x58), value: P_TextModeWrite.nRow, style: BarDisplayImage-Gray, scale format: %.1f, scale 0..100
        p518627256: Gerando ...
    Textfield (369,103 40x50), "%s", text variable: GVL.arrCVSfilter[GVL.radioEstufa].mes, input disabled if: GVL.radioData
        OnMouseClick: write the text variable via VisuDialogs.Numpad
    Textfield (423,103 70x50), "%s", text variable: GVL.arrCVSfilter[GVL.radioEstufa].ano, input disabled if: GVL.radioData
        OnMouseClick: write the text variable via VisuDialogs.Numpad
    GroupBox (551,52 200x112), "Ordem de Fabricação", input disabled if: GVL.radioOF
        Textfield (16,51 160x50), "%s", text variable: GVL.arrCVSfilter[GVL.radioEstufa].ordem, input disabled if: GVL.radioOF
            OnMouseClick: write the text variable via VisuDialogs.Numpad
        Label (13,19 80x29), "Número"
    GroupBox (794,52 200x112), "Lote", input disabled if: GVL.radioLote
        Textfield (16,51 160x50), "%s", text variable: GVL.arrCVSfilter[GVL.radioEstufa].lote, input disabled if: GVL.radioLote
            OnMouseClick: write the text variable via VisuDialogs.Keypad
        Label (12,19 52x29), "Letra"
    GroupBox (305,52 200x112), "Data", input disabled if: GVL.radioData
        Label (-13,19 80x29), "Dia"
        Label (43,20 80x29), "Mês"
        Label (97,20 80x29), "Ano"
    Button (1117,569 184x57), "Gerar Histórico"
        OnMouseClick: execute { gvl.bHistory:=true; }
END_VISUALIZATION

// ---- VISUs/IniciaProg_3.TcVIS
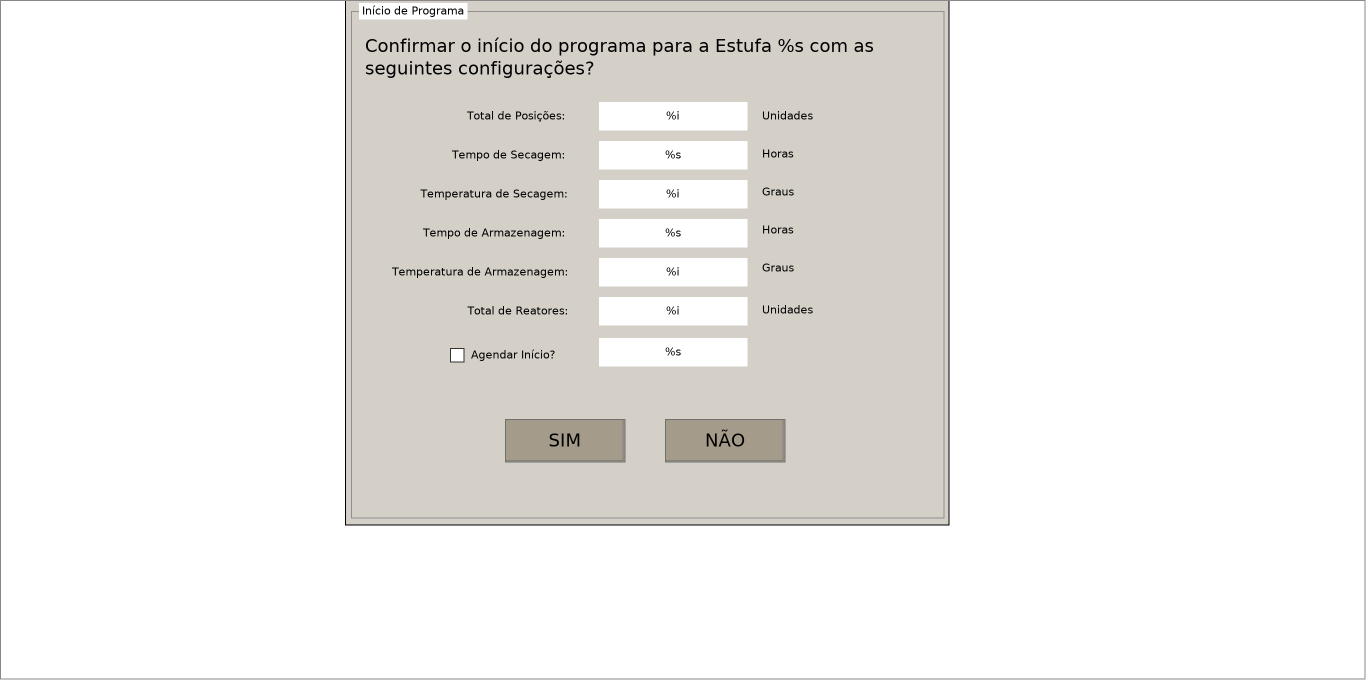
VISUALIZATION IniciaProg_3  // 1366x680
    Rectangle (345,0 604x525)
    GroupBox (351,3 593x515), "Início de Programa"
        Label (111,98 108x30), "Total de Posições:"
        Textfield (247,98 150x30), "%i", text variable: GVL.totalPos[GVL.actEst]
        Label (99,137 117x30), "Tempo de Secagem:"
        Label (65,176 156x30), "Temperatura de Secagem:"
        Label (67,215 152x30), "Tempo de Armazenagem:"
        Label (37,254 184x30), "Temperatura de Armazenagem:"
        Label (113,293 108x30), "Total de Reatores:"
        Textfield (247,137 150x30), "%s", text variable: GVL.totalSeca[2]
        Textfield (247,176 150x30), "%i", text variable: GVL_P.arrStatusEstufas[gvl.actEst].tempSeca
        Textfield (247,215 150x30), "%s", text variable: GVL.totalArm[2]
        Textfield (247,254 150x30), "%i", text variable: GVL_P.arrStatusEstufas[gvl.actEst].tempArm
        Textfield (247,293 150x30), "%i", text variable: GVL.totalRaet[GVL.actEst]
        Label (408,98 62x30), "Unidades"
        Label (408,136 62x30), "Horas"
        Label (408,174 62x30), "Graus"
        Label (408,212 62x30), "Horas"
        Label (408,250 62x30), "Graus"
        Label (408,292 62x30), "Unidades"
        Button (154,416 120x43), "SIM"
            OnMouseClick: CloseDialog Dialog=IniciaProg_3, Result=Yes, NumpadKeypadSet=True
            OnMouseClick: execute { simIniciaProg(); }
        Button (314,416 120x43), "NÃO"
            OnMouseClick: CloseDialog Dialog=IniciaProg_3, Result=No, NumpadKeypadSet=True
        Textfield (247,334 150x30), "%s", text variable: GVL.progInicio[GVL.actEst], input disabled if: not GVL.bAgendaInicio
            OnMouseClick: OpenDialog Dialog=setInicio, OpenModal=True, OpenCentered=True
            OnMouseClick: execute {
                gvl.dia:= MID(STR:= gvl.progInicio[gvl.actEst] , LEN:= 2, POS:=12);
                gvl.mes:= MID(STR:= gvl.progInicio[gvl.actEst] , LEN:= 2, POS:=9);
                gvl.ano:= MID(STR:= gvl.progInicio[gvl.actEst] , LEN:= 2, POS:=6);
                gvl.hora:= MID(STR:= gvl.progInicio[gvl.actEst] , LEN:= 2, POS:=15);
                gvl.minuto:= MID(STR:= gvl.progInicio[gvl.actEst] , LEN:= 2, POS:=18);
            }
    Checkbox (448,341 122x28), "Agendar Início?", variable: GVL.bAgendaInicio
    Rectangle (362,30 574x54), "Confirmar o início do programa para a Estufa %s com as seguintes configurações?", text variable: GVL.estAtiva
END_VISUALIZATION

// ---- VISUs/IniciaProg_2.TcVIS
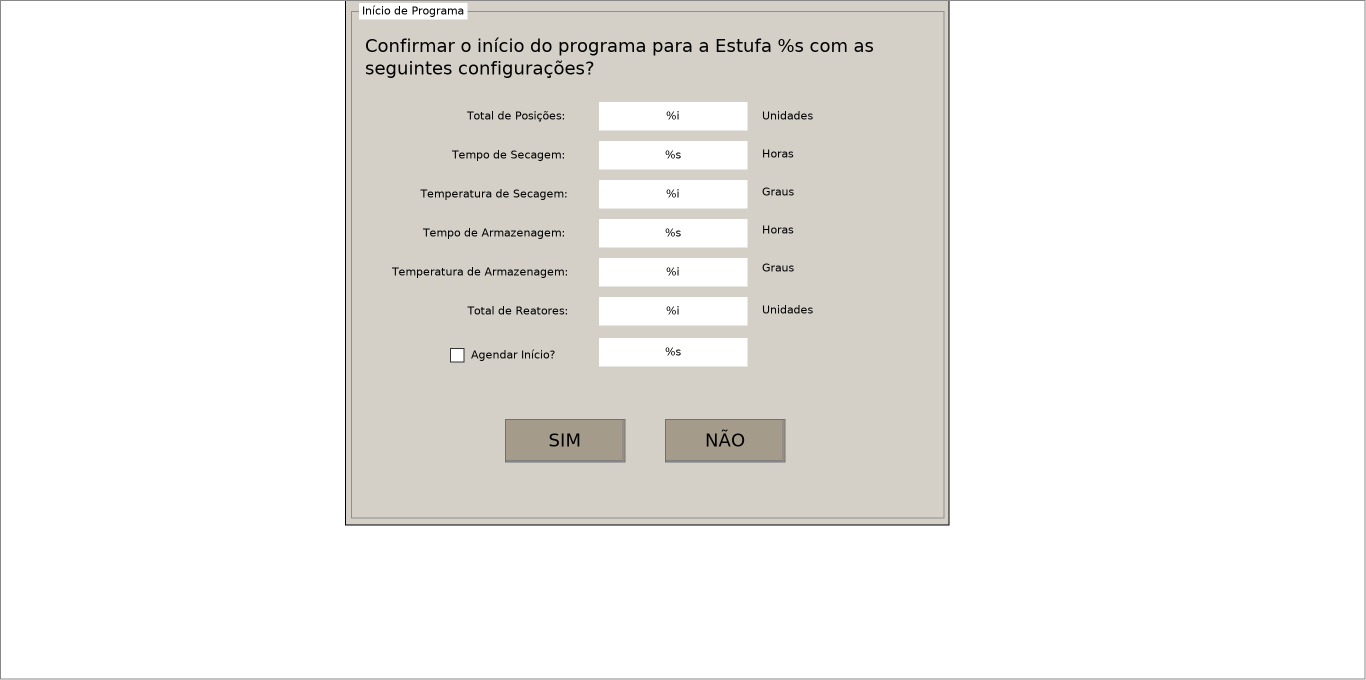
VISUALIZATION IniciaProg_2  // 1366x680
    Rectangle (345,0 604x525)
    GroupBox (351,3 593x515), "Início de Programa"
        Label (111,98 108x30), "Total de Posições:"
        Textfield (247,98 150x30), "%i", text variable: GVL.totalPos[GVL.actEst]
        Label (99,137 117x30), "Tempo de Secagem:"
        Label (65,176 156x30), "Temperatura de Secagem:"
        Label (67,215 152x30), "Tempo de Armazenagem:"
        Label (37,254 184x30), "Temperatura de Armazenagem:"
        Label (113,293 108x30), "Total de Reatores:"
        Textfield (247,137 150x30), "%s", text variable: GVL.totalSeca[GVL.actEst]
        Textfield (247,176 150x30), "%i", text variable: GVL_P.arrStatusEstufas[gvl.actEst].tempSeca
        Textfield (247,215 150x30), "%s", text variable: GVL.totalArm[GVL.actEst]
        Textfield (247,254 150x30), "%i", text variable: GVL_P.arrStatusEstufas[gvl.actEst].tempArm
        Textfield (247,293 150x30), "%i", text variable: GVL.totalRaet[GVL.actEst]
        Label (408,98 62x30), "Unidades"
        Label (408,136 62x30), "Horas"
        Label (408,174 62x30), "Graus"
        Label (408,212 62x30), "Horas"
        Label (408,250 62x30), "Graus"
        Label (408,292 62x30), "Unidades"
        Button (154,416 120x43), "SIM"
            OnMouseClick: CloseDialog Dialog=IniciaProg_2, Result=Yes, NumpadKeypadSet=True
            OnMouseClick: execute { simIniciaProg(); }
        Button (314,416 120x43), "NÃO"
            OnMouseClick: CloseDialog Dialog=IniciaProg_2, Result=No, NumpadKeypadSet=True
        Textfield (247,334 150x30), "%s", text variable: GVL.progInicio[GVL.actEst], input disabled if: not GVL.bAgendaInicio
            OnMouseClick: OpenDialog Dialog=setInicio, OpenModal=True, OpenCentered=True
            OnMouseClick: execute {
                gvl.dia:= MID(STR:= gvl.progInicio[gvl.actEst] , LEN:= 2, POS:=12);
                gvl.mes:= MID(STR:= gvl.progInicio[gvl.actEst] , LEN:= 2, POS:=9);
                gvl.ano:= MID(STR:= gvl.progInicio[gvl.actEst] , LEN:= 2, POS:=6);
                gvl.hora:= MID(STR:= gvl.progInicio[gvl.actEst] , LEN:= 2, POS:=15);
                gvl.minuto:= MID(STR:= gvl.progInicio[gvl.actEst] , LEN:= 2, POS:=18);
            }
    Checkbox (448,341 122x28), "Agendar Início?", variable: GVL.bAgendaInicio
    Rectangle (362,30 574x54), "Confirmar o início do programa para a Estufa %s com as seguintes configurações?", text variable: GVL.estAtiva
END_VISUALIZATION

// ---- VISUs/Manu021.TcVIS
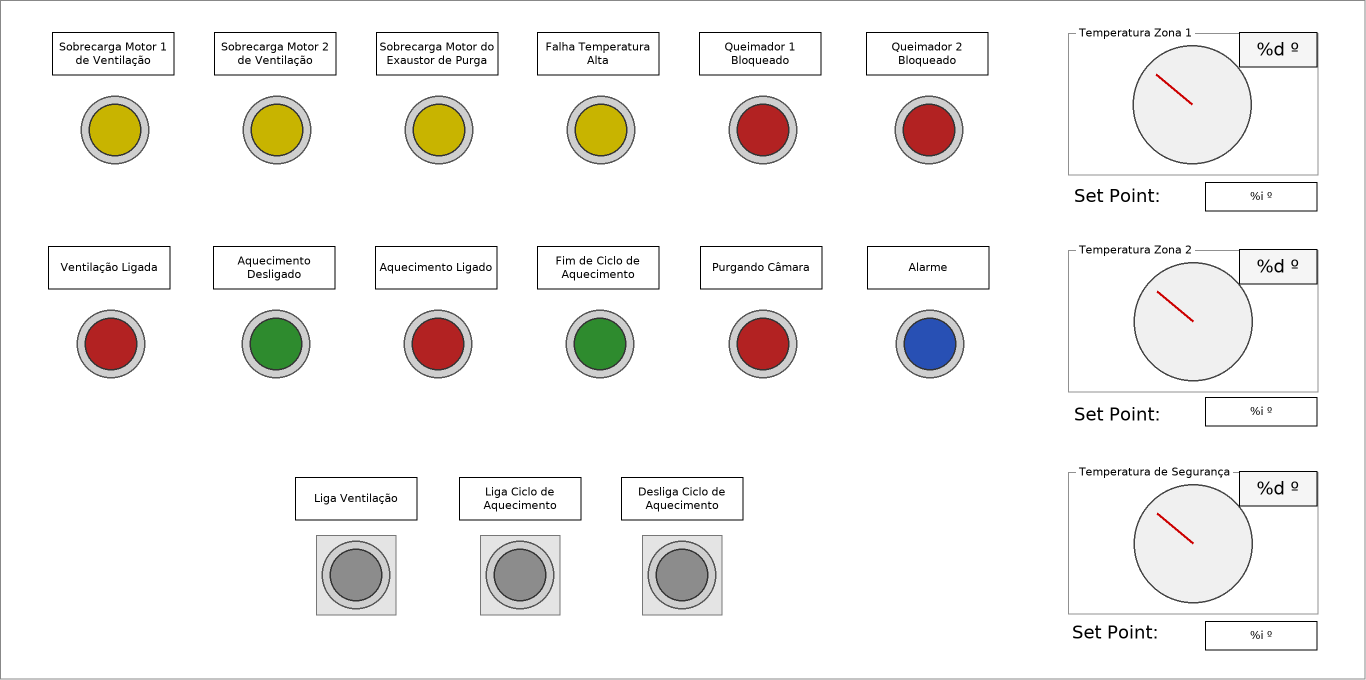
VISUALIZATION Manu021  // 1366x680
    Lamp1 (75,90 80x80), variable: GVL.sobrecarga_M1_vent_021, style: Lamp-Lamp1-Yellow
    Lamp1 (237,90 80x80), variable: GVL.sobrecarga_M2_vent_021, style: Lamp-Lamp1-Yellow
    Lamp1 (399,90 80x80), variable: GVL.sobrecarga_Purga_021, style: Lamp-Lamp1-Yellow
    Lamp1 (561,90 80x80), variable: GVL.falhaTempHigh_021, style: Lamp-Lamp1-Yellow
    Lamp1 (723,90 80x80), variable: GVL.queimador1_block_021, style: Lamp-Lamp1-Red
    Lamp1 (889,90 80x80), variable: GVL.queimador2_block_021, style: Lamp-Lamp1-Red
    Rectangle (52,32 122x43), "Sobrecarga Motor 1 de Ventilação"
    Rectangle (214,32 122x43), "Sobrecarga Motor 2 de Ventilação"
    Rectangle (376,32 122x43), "Sobrecarga Motor do Exaustor de Purga"
    Rectangle (537,32 122x43), "Falha Temperatura Alta"
    Rectangle (699,32 122x43), "Queimador 1 Bloqueado"
    Rectangle (866,32 122x43), "Queimador 2 Bloqueado"
    Lamp1 (71,304 80x80), variable: GVL.ventilacao_Ligada_021, style: Lamp-Lamp1-Red
    Rectangle (48,246 122x43), "Ventilação Ligada"
    Lamp1 (236,304 80x80), variable: GVL.aquecimento_Desligado_021, style: Lamp-Lamp1-Green
    Rectangle (213,246 122x43), "Aquecimento Desligado"
    Lamp1 (398,304 80x80), variable: GVL.aquecimento_Ligado_021, style: Lamp-Lamp1-Red
    Rectangle (375,246 122x43), "Aquecimento Ligado"
    Lamp1 (560,304 80x80), variable: GVL.fimCicloAquecimento_021, style: Lamp-Lamp1-Green
    Rectangle (537,246 122x43), "Fim de Ciclo de Aquecimento"
    Lamp1 (723,304 80x80), variable: GVL.purgandoCamara_021, style: Lamp-Lamp1-Red
    Rectangle (700,246 122x43), "Purgando Câmara"
    PushSwitch (316,535 80x80), variable: GVL.liga_ventilacao_021, behaviour: TAP, style: Switch-PushSwitch-Gray
    Rectangle (295,477 122x43), "Liga Ventilação"
    PushSwitch (480,535 80x80), variable: GVL.liga_aquecimento_021, behaviour: TAP, style: Switch-PushSwitch-Gray
    Rectangle (459,477 122x43), "Liga Ciclo de Aquecimento"
    PushSwitch (642,535 80x80), variable: GVL.desl_aquecimento_021, behaviour: TAP, style: Switch-PushSwitch-Gray
    Rectangle (621,477 122x43), "Desliga Ciclo de Aquecimento"
    Lamp1 (890,304 80x80), style: Lamp-Lamp1-Blue
    Rectangle (867,246 122x43), "Alarme"
    GroupBox (1068,25 250x150), "Temperatura Zona 1"
    Meter180 (1072,45 240x119), value: GVL.zona1atual_021, style: Meter-Meter180-Gray, scale format: %.1f, scale 20..160
        p518627256: ºC
    GroupBox (1068,242 250x150), "Temperatura Zona 2"
        Rectangle (171,7 78x35), "%d º", text variable: GVL.zona2atual_021
    Meter180 (1073,262 240x119), value: GVL.zona2atual_021, style: Meter-Meter180-Gray, scale format: %.1f, scale 20..160
        p518627256: ºC
    GroupBox (1068,464 250x150), "Temperatura de Segurança"
    Meter180 (1073,484 240x119), value: GVL.zonaSegAtual_021, style: Meter-Meter180-Gray, scale format: %.1f, scale 20..160
        p518627256: ºC
    Rectangle (1205,182 112x29), "%i º", text variable: GVL_P.zona1setpt_021
        OnMouseClick: write GVL_P.zona1setpt_021 via VisuDialogs.Numpad
    Label (1072,185 91x22), "Set Point:"
    Rectangle (1205,397 112x29), "%i º", text variable: GVL_P.zona2setpt_021
        OnMouseClick: write GVL_P.zona2setpt_021 via VisuDialogs.Numpad
    Label (1072,400 91x29), "Set Point:"
    Rectangle (1239,32 78x35), "%d º", text variable: GVL.zona1atual_021
    Rectangle (1239,471 78x35), "%d º", text variable: GVL.zonaSegAtual_021
    Label (1070,618 91x29), "Set Point:"
    Rectangle (1205,621 112x29), "%i º", text variable: GVL_P.zonaSegSetpt_021
        OnMouseClick: write GVL_P.zonaSegSetpt_021 via VisuDialogs.Numpad
END_VISUALIZATION

// ---- VISUs/Manu020.TcVIS
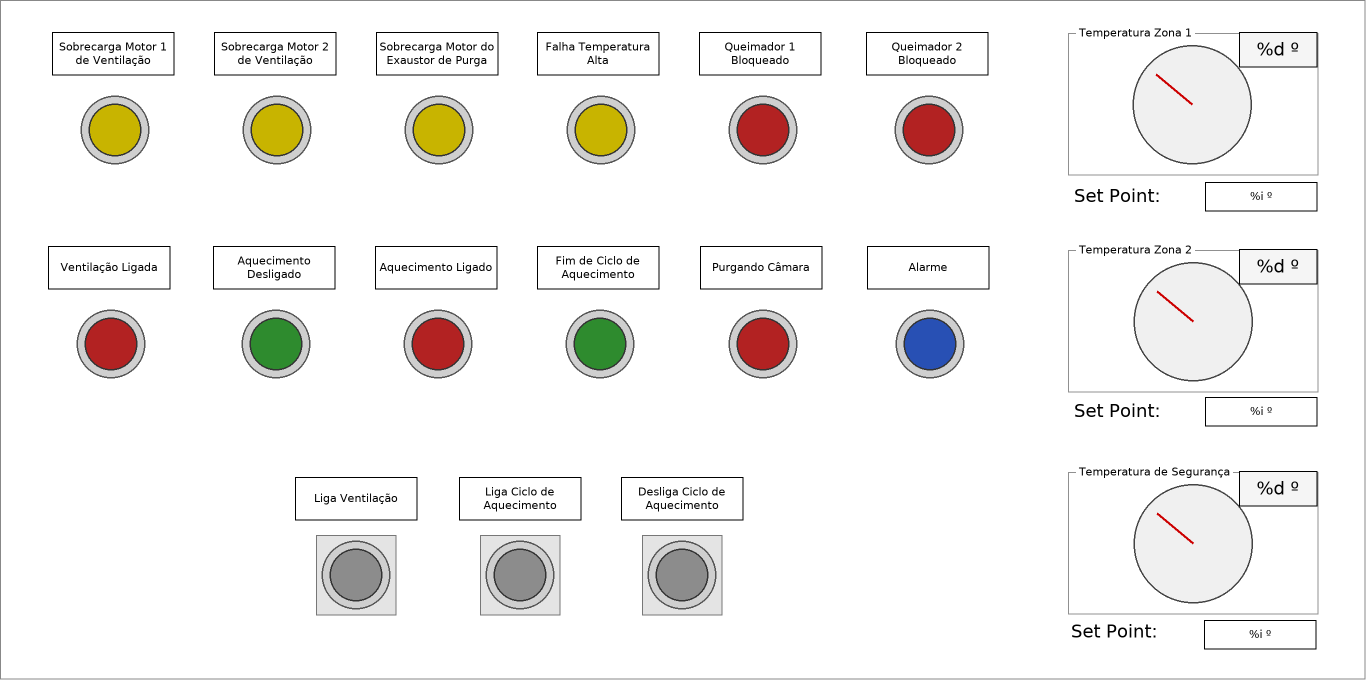
VISUALIZATION Manu020  // 1366x680
    Lamp1 (75,90 80x80), variable: GVL.sobrecarga_M1_vent_020, style: Lamp-Lamp1-Yellow
    Lamp1 (237,90 80x80), variable: GVL.sobrecarga_M2_vent_020, style: Lamp-Lamp1-Yellow
    Lamp1 (399,90 80x80), variable: GVL.sobrecarga_Purga_020, style: Lamp-Lamp1-Yellow
    Lamp1 (561,90 80x80), variable: GVL.falhaTempHigh_020, style: Lamp-Lamp1-Yellow
    Lamp1 (723,90 80x80), variable: GVL.queimador1_block_020, style: Lamp-Lamp1-Red
    Lamp1 (889,90 80x80), variable: GVL.queimador2_block_020, style: Lamp-Lamp1-Red
    Rectangle (52,32 122x43), "Sobrecarga Motor 1 de Ventilação"
    Rectangle (214,32 122x43), "Sobrecarga Motor 2 de Ventilação"
    Rectangle (376,32 122x43), "Sobrecarga Motor do Exaustor de Purga"
    Rectangle (537,32 122x43), "Falha Temperatura Alta"
    Rectangle (699,32 122x43), "Queimador 1 Bloqueado"
    Rectangle (866,32 122x43), "Queimador 2 Bloqueado"
    Lamp1 (71,304 80x80), variable: GVL.ventilacao_Ligada_020, style: Lamp-Lamp1-Red
    Rectangle (48,246 122x43), "Ventilação Ligada"
    Lamp1 (236,304 80x80), variable: GVL.aquecimento_Desligado_020, style: Lamp-Lamp1-Green
    Rectangle (213,246 122x43), "Aquecimento Desligado"
    Lamp1 (398,304 80x80), variable: GVL.aquecimento_Ligado_020, style: Lamp-Lamp1-Red
    Rectangle (375,246 122x43), "Aquecimento Ligado"
    Lamp1 (560,304 80x80), variable: GVL.fimCicloAquecimento_020, style: Lamp-Lamp1-Green
    Rectangle (537,246 122x43), "Fim de Ciclo de Aquecimento"
    Lamp1 (723,304 80x80), variable: GVL.purgandoCamara_020, style: Lamp-Lamp1-Red
    Rectangle (700,246 122x43), "Purgando Câmara"
    PushSwitch (316,535 80x80), variable: GVL.liga_ventilacao_020, behaviour: TAP, style: Switch-PushSwitch-Gray
    Rectangle (295,477 122x43), "Liga Ventilação"
    PushSwitch (480,535 80x80), variable: GVL.liga_aquecimento_020, behaviour: TAP, style: Switch-PushSwitch-Gray
    Rectangle (459,477 122x43), "Liga Ciclo de Aquecimento"
    PushSwitch (642,535 80x80), variable: GVL.desl_aquecimento_020, behaviour: TAP, style: Switch-PushSwitch-Gray
    Rectangle (621,477 122x43), "Desliga Ciclo de Aquecimento"
    Lamp1 (890,304 80x80), style: Lamp-Lamp1-Blue
    Rectangle (867,246 122x43), "Alarme"
    GroupBox (1068,25 250x150), "Temperatura Zona 1"
    Meter180 (1072,45 240x119), value: GVL.zona1atual_020, style: Meter-Meter180-Gray, scale format: %.1f, scale 20..160
        p518627256: ºC
    GroupBox (1068,242 250x150), "Temperatura Zona 2"
    Meter180 (1073,262 240x119), value: GVL.zona2atual_020, style: Meter-Meter180-Gray, scale format: %.1f, scale 20..160
        p518627256: ºC
    GroupBox (1068,464 250x150), "Temperatura de Segurança"
    Meter180 (1073,484 240x119), value: GVL.zonaSegAtual_020, style: Meter-Meter180-Gray, scale format: %.1f, scale 20..160
        p518627256: ºC
    Rectangle (1205,182 112x29), "%i º", text variable: GVL_P.zona1setpt_020
        OnMouseClick: write GVL_P.zona1setpt_020 via VisuDialogs.Numpad
    Label (1072,185 91x22), "Set Point:"
    Rectangle (1205,397 112x29), "%i º", text variable: GVL_P.zona2setpt_020
        OnMouseClick: write GVL_P.zona2setpt_020 via VisuDialogs.Numpad
    Label (1072,400 91x22), "Set Point:"
    Rectangle (1239,32 78x35), "%d º", text variable: GVL.zona1atual_020
    Rectangle (1239,249 78x35), "%d º", text variable: GVL.zona2atual_020
    Label (1069,617 91x29), "Set Point:"
    Rectangle (1204,620 112x29), "%i º", text variable: GVL_P.zonaSegSetpt_020
        OnMouseClick: write the text variable via VisuDialogs.Numpad
    Rectangle (1239,471 78x35), "%d º", text variable: GVL.zonaSegAtual_020
END_VISUALIZATION

// ---- VISUs/Notifica24horas.TcVIS
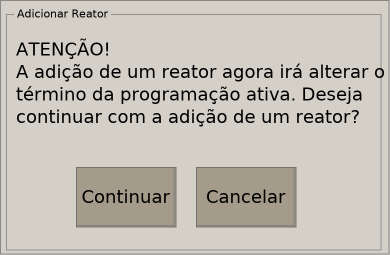
VISUALIZATION Notifica24horas  // 390x255
    GroupBox (6,6 375x244), "Adicionar Reator"
        Label (7,31 373x126), "ATENÇÃO! A adição de um reator agora irá alterar o término da programação ativa. Deseja continuar com a adição de um reator?"
        Button (70,161 100x60), "Continuar"
            OnMouseClick: execute {
                posCarrinho.bNotificaTime:=TRUE;
                posCarrinho2.bNotificaTime:=TRUE;
                posCarrinho3.bNotificaTime:=TRUE;
            }
        Button (190,161 100x60), "Cancelar"
            OnMouseClick: CloseDialog Dialog=ConfigPosicao_Reator, Result=Cancel, NumpadKeypadSet=True
            OnMouseClick: execute {
                posCarrinho.bNotificaTime:=TRUE;
                posCarrinho2.bNotificaTime:=TRUE;
                posCarrinho3.bNotificaTime:=TRUE;
            }
            OnMouseClick: CloseDialog Dialog=ConfigPosicao_Reator_2, Result=Cancel, NumpadKeypadSet=True
            OnMouseClick: CloseDialog Dialog=ConfigPosicao_Reator_3, Result=Cancel, NumpadKeypadSet=True
END_VISUALIZATION

// ---- VISUs/Manu019.TcVIS
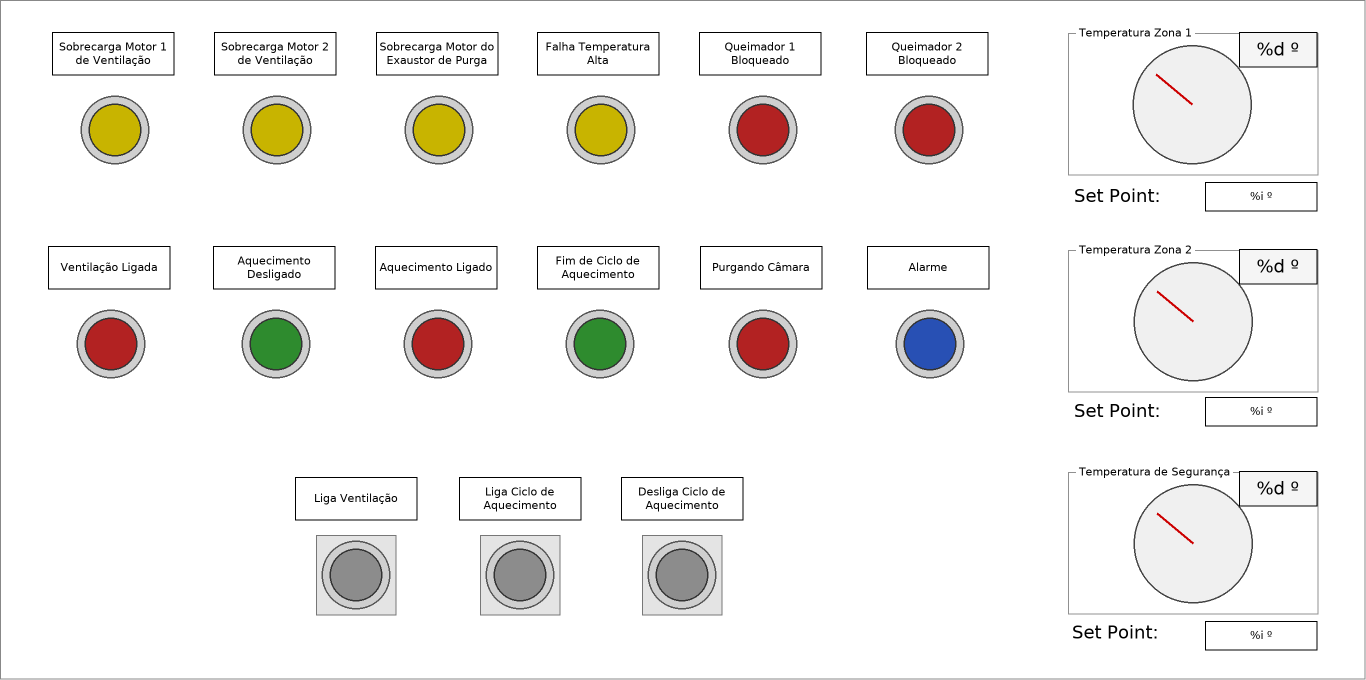
VISUALIZATION Manu019  // 1366x680
    Lamp1 (75,90 80x80), variable: GVL.sobrecarga_M1_vent_019, style: Lamp-Lamp1-Yellow
    Lamp1 (237,90 80x80), variable: GVL.sobrecarga_M2_vent_019, style: Lamp-Lamp1-Yellow
    Lamp1 (399,90 80x80), variable: GVL.sobrecarga_Purga_019, style: Lamp-Lamp1-Yellow
    Lamp1 (561,90 80x80), variable: GVL.falhaTempHigh_019, style: Lamp-Lamp1-Yellow
    Lamp1 (723,90 80x80), variable: GVL.queimador1_block_019, style: Lamp-Lamp1-Red
    Lamp1 (889,90 80x80), variable: GVL.queimador2_block_019, style: Lamp-Lamp1-Red
    Rectangle (52,32 122x43), "Sobrecarga Motor 1 de Ventilação"
    Rectangle (214,32 122x43), "Sobrecarga Motor 2 de Ventilação"
    Rectangle (376,32 122x43), "Sobrecarga Motor do Exaustor de Purga"
    Rectangle (537,32 122x43), "Falha Temperatura Alta"
    Rectangle (699,32 122x43), "Queimador 1 Bloqueado"
    Rectangle (866,32 122x43), "Queimador 2 Bloqueado"
    Lamp1 (71,304 80x80), variable: GVL.ventilacao_Ligada_019, style: Lamp-Lamp1-Red
    Rectangle (48,246 122x43), "Ventilação Ligada"
    Lamp1 (236,304 80x80), variable: GVL.aquecimento_Desligado_019, style: Lamp-Lamp1-Green
    Rectangle (213,246 122x43), "Aquecimento Desligado"
    Lamp1 (398,304 80x80), variable: GVL.aquecimento_Ligado_019, style: Lamp-Lamp1-Red
    Rectangle (375,246 122x43), "Aquecimento Ligado"
    Lamp1 (560,304 80x80), variable: GVL.fimCicloAquecimento_019, style: Lamp-Lamp1-Green
    Rectangle (537,246 122x43), "Fim de Ciclo de Aquecimento"
    Lamp1 (723,304 80x80), variable: GVL.purgandoCamara_019, style: Lamp-Lamp1-Red
    Rectangle (700,246 122x43), "Purgando Câmara"
    PushSwitch (316,535 80x80), variable: GVL.liga_ventilacao_019, behaviour: TAP, style: Switch-PushSwitch-Gray
    Rectangle (295,477 122x43), "Liga Ventilação"
    PushSwitch (480,535 80x80), variable: GVL.liga_aquecimento_019, behaviour: TAP, style: Switch-PushSwitch-Gray
    Rectangle (459,477 122x43), "Liga Ciclo de Aquecimento"
    PushSwitch (642,535 80x80), variable: GVL.desl_aquecimento_019, behaviour: TAP, style: Switch-PushSwitch-Gray
    Rectangle (621,477 122x43), "Desliga Ciclo de Aquecimento"
    Lamp1 (890,304 80x80), style: Lamp-Lamp1-Blue
    Rectangle (867,246 122x43), "Alarme"
    GroupBox (1068,25 250x150), "Temperatura Zona 1"
    Meter180 (1072,45 240x119), value: GVL.zona1atual_019, style: Meter-Meter180-Gray, scale format: %.1f, scale 20..160
        p518627256: ºC
    GroupBox (1068,242 250x150), "Temperatura Zona 2"
    Meter180 (1073,262 240x119), value: GVL.zona2atual_019, style: Meter-Meter180-Gray, scale format: %.1f, scale 20..160
        p518627256: ºC
    GroupBox (1068,464 250x150), "Temperatura de Segurança"
    Meter180 (1073,484 240x119), value: GVL.zonaSegAtual_019, style: Meter-Meter180-Gray, scale format: %.1f, scale 20..160
        p518627256: ºC
    Rectangle (1205,182 112x29), "%i º", text variable: GVL_P.zona1setpt_019
        OnMouseClick: write GVL_P.zona1setpt_019 via VisuDialogs.Numpad
    Label (1072,185 91x22), "Set Point:"
    Rectangle (1205,397 112x29), "%i º", text variable: GVL_P.zona2setpt_019
        OnMouseClick: write GVL_P.zona2setpt_019 via VisuDialogs.Numpad
    Label (1072,400 91x22), "Set Point:"
    Rectangle (1239,32 78x35), "%d º", text variable: GVL.zona1atual_019
    Rectangle (1239,249 78x35), "%d º", text variable: GVL.zona2atual_019
    Rectangle (1239,471 78x35), "%d º", text variable: GVL.zonaSegAtual_019
    Label (1070,618 91x29), "Set Point:"
    Rectangle (1205,621 112x29), "%i º", text variable: GVL_P.zonaSegSetpt_019
        OnMouseClick: write the text variable via VisuDialogs.Numpad
END_VISUALIZATION

// ---- VISUs/Carrinho.TcVIS
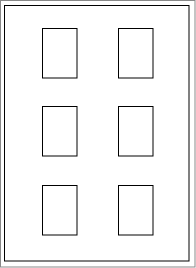
VISUALIZATION Carrinho  // 196x268
    RoundedRectangle (4,5 185x256)
    RoundedRectangle (35,36 50x35), angle 90, colour variable: GVL_P.corPosReator1[4].color
        OnMouseUp: execute { gvl.actReat:= 4; }
        OnMouseUp: OpenDialog Dialog=ConfigPosicao_Reator, Parameters={bReator: , iOFnumber: , iSrlNumber: }, OpenModal=True, OpenCentered=True
    RoundedRectangle (111,36 50x35), angle 90, colour variable: GVL_P.corPosReator1[1].color
        OnMouseUp: OpenDialog Dialog=ConfigPosicao_Reator, Parameters={bReator: , iOFnumber: , iSrlNumber: }, OpenModal=True, OpenCentered=True
        OnMouseUp: execute { gvl.actReat:= 1; posCarrinho(); }
    RoundedRectangle (111,114 50x35), angle 90, colour variable: GVL_P.corPosReator1[2].color
        OnMouseUp: execute { gvl.actReat:= 2; }
        OnMouseUp: OpenDialog Dialog=ConfigPosicao_Reator, Parameters={bReator: , iOFnumber: , iSrlNumber: }, OpenModal=True, OpenCentered=True
    RoundedRectangle (35,114 50x35), angle 90, colour variable: GVL_P.corPosReator1[5].color
        OnMouseUp: execute { gvl.actReat:= 5; }
        OnMouseUp: OpenDialog Dialog=ConfigPosicao_Reator, Parameters={bReator: , iOFnumber: , iSrlNumber: }, OpenModal=True, OpenCentered=True
    RoundedRectangle (111,193 50x35), angle 90, colour variable: GVL_P.corPosReator1[3].color
        OnMouseUp: execute { gvl.actReat:= 3; }
        OnMouseUp: OpenDialog Dialog=ConfigPosicao_Reator, Parameters={bReator: , iOFnumber: , iSrlNumber: }, OpenModal=True, OpenCentered=True
    RoundedRectangle (35,193 50x35), angle 90, colour variable: GVL_P.corPosReator1[6].color
        OnMouseUp: execute { gvl.actReat:= 6; }
        OnMouseUp: OpenDialog Dialog=ConfigPosicao_Reator, Parameters={bReator: , iOFnumber: , iSrlNumber: }, OpenModal=True, OpenCentered=True
END_VISUALIZATION

// ---- VISUs/Estufa1.TcVIS
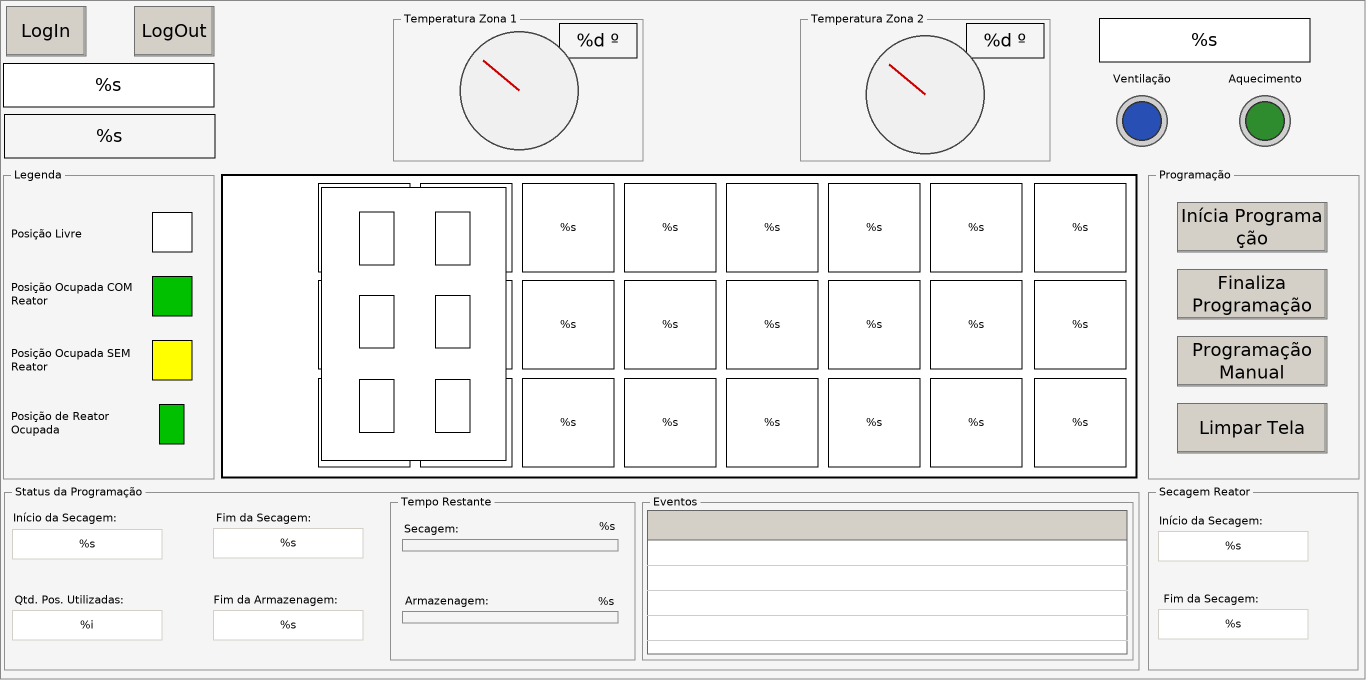
VISUALIZATION Estufa1  // 1366x680
    GroupBox (1148,484 210x186), "Secagem Reator", invisible if: GVL_P.bCarrinhoReator1
        Label (10,100 106x30), "Fim da Secagem:"
        Textfield (10,125 150x30), "%s", text variable: GVL_P.arrStatusEstufas[0].statusFimSecagem
    GroupBox (3,167 211x312), "Legenda"
        RoundedRectangle (149,173 40x40)
        RoundedRectangle (149,45 40x40)
        RoundedRectangle (156,237 25x40)
    GroupBox (800,11 250x150), "Temperatura Zona 2"
        Rectangle (166,12 78x35), "%d º", text variable: GVL.zona2atual_019
    GroupBox (393,11 250x150), "Temperatura Zona 1"
        Rectangle (166,12 78x35), "%d º", text variable: GVL.zona1atual_019
    GroupBox (4,484 1135x186), "Status da Programação"
        Label (209,19 101x30), "Fim da Secagem:"
        Label (209,101 125x30), "Fim da Armazenagem:"
        Label (8,101 114x30), "Qtd. Pos. Utilizadas:"
        GroupBox (638,10 491x166), "Eventos"
            Table (5,16 480x144), data array: GVL_P.arrLogEstufa19
                p3854506369: GVL_P.arrLogEstufa19[INDEX]
            InvisibleInput (6,17 431x142)
                OnMouseClick: OpenDialog Dialog=addComment, OpenModal=True, OpenCentered=True
        Label (8,19 106x30), "Início da Secagem:"
        Textfield (8,126 150x30), "%i", text variable: GVL.totalPos[0]
        Textfield (209,44 150x30), "%s", text variable: GVL_P.arrStatusEstufas[0].statusFimSecagem
        Textfield (209,126 150x30), "%s", text variable: GVL_P.arrStatusEstufas[0].statusFimArmazenagem
        GroupBox (386,10 245x166), "Tempo Restante"
            Progressbar (12,117 216x12), variable: MAIN.bardintArm19
            Rectangle (131,99 96x17), "%s", text variable: mid(str:=time_to_string(GVL.endArm19), LEN:= 20, POS:= 3)
            Progressbar (12,45 216x12), variable: MAIN.bardintSec19
        Label (398,30 59x30), "Secagem:"
    Rectangle (221,174 916x304)
    Rectangle (1034,183 92x89), "%s", text variable: GVL_P.aPositionsE019[1].text, colour variable: GVL_P.aPositionsE019[1].color
        OnMouseUp: OpenDialog Dialog=ConfigPosicao, Parameters={bReator: , iOFnumber: , iSrlNumber: }, OpenModal=True, OpenCentered=True
        OnMouseUp: execute {
            gvl.actPos:= 1;
            //selectPos019();
        }
    Rectangle (1034,280 92x89), "%s", text variable: GVL_P.aPositionsE019[2].text, colour variable: GVL_P.aPositionsE019[2].color
        OnMouseUp: OpenDialog Dialog=ConfigPosicao, Parameters={bReator: , iOFnumber: , iSrlNumber: }, OpenModal=True, OpenCentered=True
        OnMouseUp: execute {
            gvl.actPos:= 2;
            //selectPos019();
        }
    Rectangle (1034,378 92x89), "%s", text variable: GVL_P.aPositionsE019[3].text, colour variable: GVL_P.aPositionsE019[3].color
        OnMouseUp: OpenDialog Dialog=ConfigPosicao, Parameters={bReator: , iOFnumber: , iSrlNumber: }, OpenModal=True, OpenCentered=True
        OnMouseUp: execute {
            gvl.actPos:= 3;
            //selectPos019();
        }
    Rectangle (930,183 92x89), "%s", text variable: GVL_P.aPositionsE019[4].text, colour variable: GVL_P.aPositionsE019[4].color
        OnMouseUp: OpenDialog Dialog=ConfigPosicao, Parameters={bReator: , iOFnumber: , iSrlNumber: }, OpenModal=True, OpenCentered=True
        OnMouseUp: execute {
            gvl.actPos:= 4;
            //selectPos019();
        }
    Rectangle (930,280 92x89), "%s", text variable: GVL_P.aPositionsE019[5].text, colour variable: GVL_P.aPositionsE019[5].color
        OnMouseUp: OpenDialog Dialog=ConfigPosicao, Parameters={bReator: , iOFnumber: , iSrlNumber: }, OpenModal=True, OpenCentered=True
        OnMouseUp: execute {
            gvl.actPos:= 5;
            //selectPos019();
        }
    Rectangle (930,378 92x89), "%s", text variable: GVL_P.aPositionsE019[6].text, colour variable: GVL_P.aPositionsE019[6].color
        OnMouseUp: OpenDialog Dialog=ConfigPosicao, Parameters={bReator: , iOFnumber: , iSrlNumber: }, OpenModal=True, OpenCentered=True
        OnMouseUp: execute {
            gvl.actPos:= 6;
            //selectPos019();
        }
    Rectangle (828,183 92x89), "%s", text variable: GVL_P.aPositionsE019[7].text, colour variable: GVL_P.aPositionsE019[7].color
        OnMouseUp: OpenDialog Dialog=ConfigPosicao, Parameters={bReator: , iOFnumber: , iSrlNumber: }, OpenModal=True, OpenCentered=True
        OnMouseUp: execute {
            gvl.actPos:= 7;
            //selectPos019();
        }
    Rectangle (828,280 92x89), "%s", text variable: GVL_P.aPositionsE019[8].text, colour variable: GVL_P.aPositionsE019[8].color
        OnMouseUp: OpenDialog Dialog=ConfigPosicao, Parameters={bReator: , iOFnumber: , iSrlNumber: }, OpenModal=True, OpenCentered=True
        OnMouseUp: execute {
            gvl.actPos:= 8;
            //selectPos019();
        }
    Rectangle (828,378 92x89), "%s", text variable: GVL_P.aPositionsE019[9].text, colour variable: GVL_P.aPositionsE019[9].color
        OnMouseUp: OpenDialog Dialog=ConfigPosicao, Parameters={bReator: , iOFnumber: , iSrlNumber: }, OpenModal=True, OpenCentered=True
        OnMouseUp: execute {
            gvl.actPos:= 9;
            //selectPos019();
        }
    Rectangle (726,183 92x89), "%s", text variable: GVL_P.aPositionsE019[10].text, colour variable: GVL_P.aPositionsE019[10].color
        OnMouseUp: OpenDialog Dialog=ConfigPosicao, Parameters={bReator: , iOFnumber: , iSrlNumber: }, OpenModal=True, OpenCentered=True
        OnMouseUp: execute {
            gvl.actPos:= 10;
            //selectPos019();
        }
    Rectangle (726,280 92x89), "%s", text variable: GVL_P.aPositionsE019[11].text, colour variable: GVL_P.aPositionsE019[11].color
        OnMouseUp: OpenDialog Dialog=ConfigPosicao, Parameters={bReator: , iOFnumber: , iSrlNumber: }, OpenModal=True, OpenCentered=True
        OnMouseUp: execute {
            gvl.actPos:= 11;
            //selectPos019();
        }
    Rectangle (726,378 92x89), "%s", text variable: GVL_P.aPositionsE019[12].text, colour variable: GVL_P.aPositionsE019[12].color
        OnMouseUp: OpenDialog Dialog=ConfigPosicao, Parameters={bReator: , iOFnumber: , iSrlNumber: }, OpenModal=True, OpenCentered=True
        OnMouseUp: execute {
            gvl.actPos:= 12;
            //selectPos019();
        }
    Rectangle (624,183 92x89), "%s", text variable: GVL_P.aPositionsE019[13].text, colour variable: GVL_P.aPositionsE019[13].color
        OnMouseUp: OpenDialog Dialog=ConfigPosicao, Parameters={bReator: , iOFnumber: , iSrlNumber: }, OpenModal=True, OpenCentered=True
        OnMouseUp: execute {
            gvl.actPos:= 13;
            //selectPos019();
        }
    Rectangle (624,280 92x89), "%s", text variable: GVL_P.aPositionsE019[14].text, colour variable: GVL_P.aPositionsE019[14].color
        OnMouseUp: OpenDialog Dialog=ConfigPosicao, Parameters={bReator: , iOFnumber: , iSrlNumber: }, OpenModal=True, OpenCentered=True
        OnMouseUp: execute {
            gvl.actPos:= 14;
            //selectPos019();
        }
    Rectangle (624,378 92x89), "%s", text variable: GVL_P.aPositionsE019[15].text, colour variable: GVL_P.aPositionsE019[15].color
        OnMouseUp: OpenDialog Dialog=ConfigPosicao, Parameters={bReator: , iOFnumber: , iSrlNumber: }, OpenModal=True, OpenCentered=True
        OnMouseUp: execute {
            gvl.actPos:= 15;
            //selectPos019();
        }
    Rectangle (522,183 92x89), "%s", text variable: GVL_P.aPositionsE019[16].text, colour variable: GVL_P.aPositionsE019[16].color
        OnMouseUp: OpenDialog Dialog=ConfigPosicao, Parameters={bReator: , iOFnumber: , iSrlNumber: }, OpenModal=True, OpenCentered=True
        OnMouseUp: execute {
            gvl.actPos:= 16;
            //selectPos019();
        }
    Rectangle (522,280 92x89), "%s", text variable: GVL_P.aPositionsE019[17].text, colour variable: GVL_P.aPositionsE019[17].color
        OnMouseUp: OpenDialog Dialog=ConfigPosicao, Parameters={bReator: , iOFnumber: , iSrlNumber: }, OpenModal=True, OpenCentered=True
        OnMouseUp: execute {
            gvl.actPos:= 17;
            //selectPos019();
        }
    Rectangle (522,378 92x89), "%s", text variable: GVL_P.aPositionsE019[18].text, colour variable: GVL_P.aPositionsE019[18].color
        OnMouseUp: OpenDialog Dialog=ConfigPosicao, Parameters={bReator: , iOFnumber: , iSrlNumber: }, OpenModal=True, OpenCentered=True
        OnMouseUp: execute {
            gvl.actPos:= 18;
            //selectPos019();
        }
    Rectangle (420,183 92x89), "%s", text variable: GVL_P.aPositionsE019[19].text, colour variable: GVL_P.aPositionsE019[19].color
        OnMouseUp: OpenDialog Dialog=ConfigPosicao, Parameters={bReator: , iOFnumber: , iSrlNumber: }, OpenModal=True, OpenCentered=True
        OnMouseUp: execute {
            gvl.actPos:= 19;
            //selectPos019();
        }
    Rectangle (420,280 92x89), "%s", text variable: GVL_P.aPositionsE019[20].text, colour variable: GVL_P.aPositionsE019[20].color
        OnMouseUp: OpenDialog Dialog=ConfigPosicao, Parameters={bReator: , iOFnumber: , iSrlNumber: }, OpenModal=True, OpenCentered=True
        OnMouseUp: execute {
            gvl.actPos:= 20;
            //selectPos019();
        }
    Rectangle (420,378 92x89), "%s", text variable: GVL_P.aPositionsE019[21].text, colour variable: GVL_P.aPositionsE019[21].color
        OnMouseUp: OpenDialog Dialog=ConfigPosicao, Parameters={bReator: , iOFnumber: , iSrlNumber: }, OpenModal=True, OpenCentered=True
        OnMouseUp: execute {
            gvl.actPos:= 21;
            //selectPos019();
        }
    Rectangle (318,183 92x89), "%s", text variable: GVL_P.aPositionsE019[22].text, colour variable: GVL_P.aPositionsE019[22].color
        OnMouseUp: OpenDialog Dialog=ConfigPosicao, Parameters={bReator: , iOFnumber: , iSrlNumber: }, OpenModal=True, OpenCentered=True
        OnMouseUp: execute {
            gvl.actPos:= 22;
            //selectPos019();
        }
    Rectangle (318,280 92x89), "%s", text variable: GVL_P.aPositionsE019[23].text, colour variable: GVL_P.aPositionsE019[23].color
        OnMouseUp: OpenDialog Dialog=ConfigPosicao, Parameters={bReator: , iOFnumber: , iSrlNumber: }, OpenModal=True, OpenCentered=True
        OnMouseUp: execute {
            gvl.actPos:= 23;
            //selectPos019();
        }
    Rectangle (318,378 92x89), "%s", text variable: GVL_P.aPositionsE019[24].text, colour variable: GVL_P.aPositionsE019[24].color
        OnMouseUp: OpenDialog Dialog=ConfigPosicao, Parameters={bReator: , iOFnumber: , iSrlNumber: }, OpenModal=True, OpenCentered=True
        OnMouseUp: execute {
            gvl.actPos:= 24;
            //selectPos019();
        }
    Meter180 (399,31 240x119), value: GVL.zona1atual_019, style: Meter-Meter180-Gray, scale format: %.1f, scale 20..160
        p518627256: ºC
    GroupBox (1148,167 211x312), "Programação"
        Button (29,35 150x50), "Inícia Programação", input disabled if: GVL_P.arrStatusEstufas[GVL.actEst].start
            OnMouseClick: OpenDialog Dialog=IniciaProg, OpenModal=True, OpenCentered=True
            OnMouseClick: execute { iniciaProgramacaoEstufa(); }
        Button (29,102 150x50), "Finaliza Programação"
            OnMouseClick: OpenDialog Dialog=FinalizaProg, Parameters={bReator: , iOFnumber: , iSrlNumber: }, OpenModal=True, OpenCentered=True
        Button (29,169 150x50), "Programação Manual", input disabled if: GVL_P.arrStatusEstufas[GVL.actEst].start
            OnMouseClick: OpenDialog Dialog=TimeCustom, OpenModal=True, OpenCentered=True
            OnMouseClick: execute { iniciaProgramacaoEstufa(); }
    Textfield (12,529 150x30), "%s", text variable: GVL_P.arrStatusEstufas[0].statusInicioSecagem
    Label (402,586 90x30), "Armazenagem:"
    Meter180 (805,35 240x119), value: GVL.zona2atual_019, style: Meter-Meter180-Gray, scale format: %.1f, scale 20..160
        p518627256: ºC
    RoundedRectangle (152,276 40x40)
    Label (8,278 132x32), "Posição Ocupada COM Reator"
    Label (8,344 128x32), "Posição Ocupada SEM Reator"
    Label (8,218 84x32), "Posição Livre"
    Label (8,407 128x32), "Posição de Reator Ocupada"
    Frame (317,182 196x286), invisible if: GVL_P.bCarrinhoReator1
        shows Carrinho()
    Rectangle (3,63 211x44), "%s", text variable: MAIN.sDB_Operador
    Lamp1 (1112,91 60x60), variable: GVL.ventilacao_Ligada_019, style: Lamp-Lamp1-Blue
    Lamp1 (1235,91 60x60), variable: GVL.aquecimento_Ligado_019, style: Lamp-Lamp1-Green
    Label (1108,64 68x30), "Ventilação"
    Label (1227,64 76x30), "Aquecimento"
    Textfield (1158,531 150x30), "%s", text variable: GVL_P.arrStatusEstufas[0].inicioReator, invisible if: GVL_P.bCarrinhoReator1
    Label (1158,506 106x30), "Início da Secagem:", invisible if: GVL_p.bCarrinhoReator1
    Rectangle (1099,18 211x44), "%s", text variable: GVL_P.etapa_process[GVL.actEst]
    Rectangle (522,518 96x17), "%s", text variable: mid(str:=time_to_string(GVL.endSeca19), LEN:= 20, POS:= 3)
    Rectangle (4,114 211x44), "%s", text variable: GVL.sSystemTime
    Button (1177,403 150x50), "Limpar Tela"
        OnMouseClick: execute {
            FOR gvl.i:=1 TO 24 BY 1 DO
            gvl_p.aPositionsE019[gvl.i].numOF:='';
            gvl_p.aPositionsE019[gvl.i].lote:='';
            gvl_p.aPositionsE019[gvl.i].class:=0;
            gvl_p.aPositionsE019[gvl.i].pot:=0;
            gvl_p.aPositionsE019[gvl.i].cor:=0;
            gvl_p.aPositionsE019[gvl.i].text:='';
            gvl_p.aPositionsE019[gvl.i].reator:=true;
            END_FOR
            FOR gvl.i:=1 TO 18 BY 1 DO
            gvl_p.corPosReator1[gvl.i].cor:=0;
            END_FOR
            gravarConfigPosicao.bReator[0]:= false;
            ///// GERADOR DE LOG -------------------------------------------------------------
            gvl.envialog:= 'Todas as posições foram limpas. ESTUFA 19';
            gvl.logRegister19:= gvl.envialog;
            gvl.sCmdInsertLog:= 'INSERT INTO [dbo].[LogGeneral] ([HistoricalTime],[Description])VALUES($'$',$'$')';
            gvl.sCmdInsertLog:= insert(gvl.sCmdInsertLog,gvl.logRegister19,74);
            gvl.sCmdInsertLog:= insert(gvl.sCmdInsertLog,gvl.sSystemDateTime,71);
            gvl.bInsertLog:= TRUE;
        }
    Button (6,6 80x50), "LogIn"
        OnMouseClick: VisuUserMgmt Type=Login
        OnMouseClick: execute { gvl.logButton:= true; }
    Button (134,6 80x50), "LogOut"
        OnMouseClick: VisuUserMgmt Type=Logout
        OnMouseClick: execute { gvl.logButton:= false; }
END_VISUALIZATION

// ---- VISUs/Grafico.TcVIS
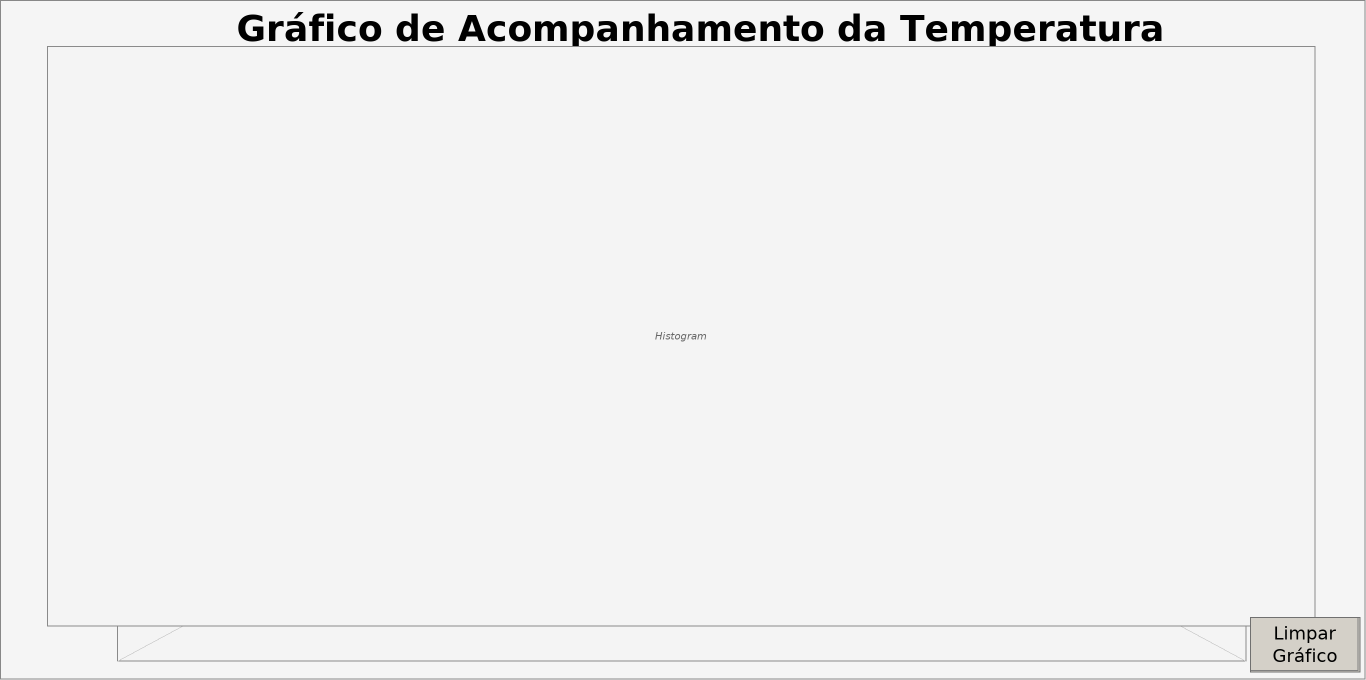
VISUALIZATION Grafico  // 1366x680
    Image (117,52 1129x609), image: ImagePool.Screenshot_3
    Histogram (47,46 1268x580), scale format: %.1f, scale 0..150
        p1518820177: GVL_P.arrTempVisu019
        p102497268: GVL_P.arrTempVisu019
        p788070771: ARRAY [1..720] OF REAL
    Label (262,7 877x43), "Gráfico de Acompanhamento da Temperatura"
    Histogram (47,46 1268x580), scale format: %.1f, scale 0..150
        p1518820177: GVL_P.arrTemp019
        p102497268: GVL_P.arrTemp019
        p788070771: ARRAY [1..720] OF REAL
    Button (1250,617 110x55), "Limpar Gráfico"
        OnMouseClick: execute {
            FOR gvl.i:=0 TO 720 BY 1 DO
            	gvl_p.arrTemp019[gvl.i]:= 0;
            	gvl_p.arrTempVisu019[gvl.i]:= 0;
            	END_FOR
        }
    InvisibleInput (831,11 54x36)
END_VISUALIZATION

// ---- VISUs/Home.TcVIS
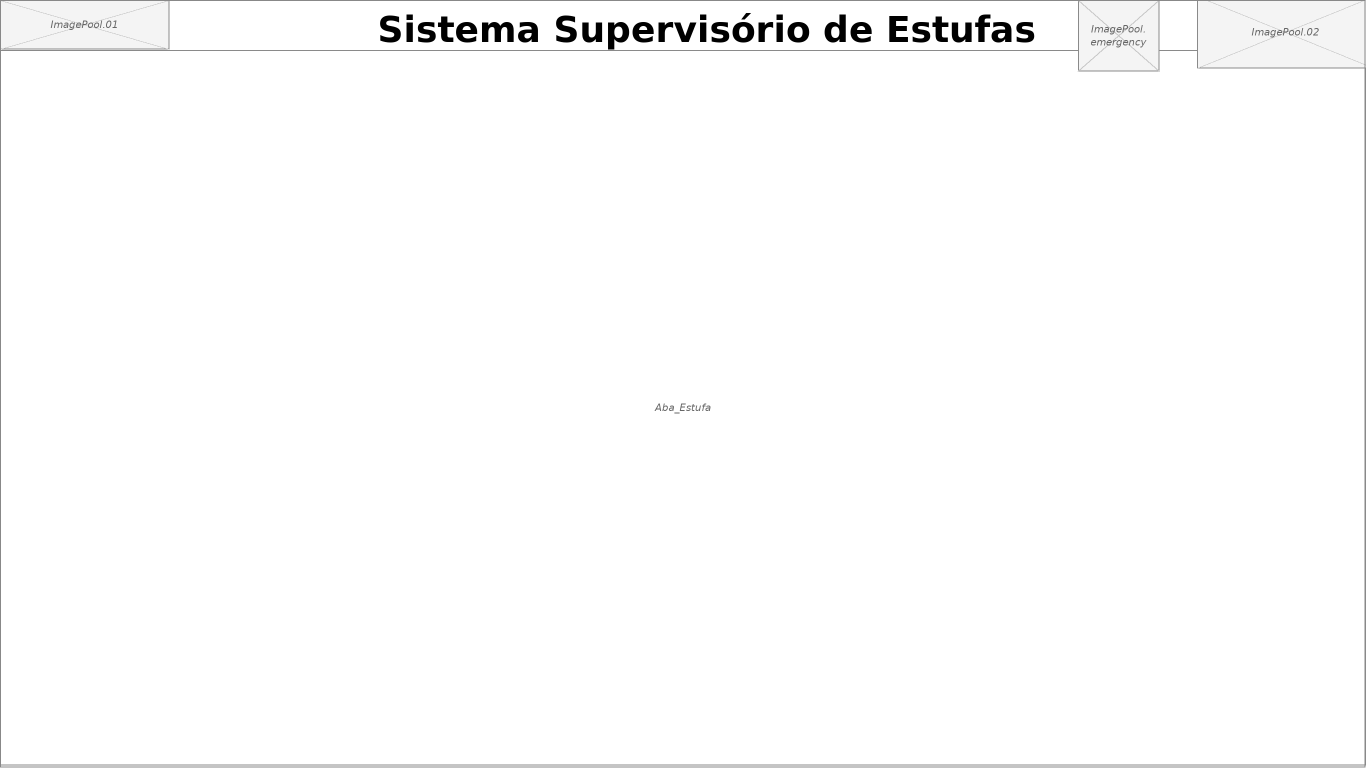
VISUALIZATION Home  // 1366x768
    TabControl (0,50 1366x715), frame switch variable: GVL.actEst
        shows Aba_Estufa()
        shows Aba_Estufa_2()
        shows Aba_Estufa_3()
        shows Aba_Manu()
        shows Historical()
        [0]: TabTitle=Estufa 203/019
        [1]: TabTitle=Estufa 203/020
        [2]: TabTitle=Estufa 203/021
        [3]: TabTitle=Manutenção
        [4]: TabTitle=Histórico
    Image (1197,-4 177x72), image: ImagePool.02
    Label (390,2 634x55), "Sistema Supervisório de Estufas"
    Image (0,0 169x49), image: ImagePool.01
    Image (1078,0 81x71), invisible if: not GVL.emergency, image: ImagePool.emergency
        OnMouseClick: execute {
            gvl.emergencia019:= FALSE;
            gvl.emergencia020:= FALSE;
            gvl.emergencia021:= FALSE;
            gvl.pwEmerg_019:= FALSE;
            gvl.pwEmerg_020:= FALSE;
            gvl.pwEmerg_021:= FALSE;
            gvl.emergency:= false;
        }
END_VISUALIZATION

// ---- VISUs/ConfigPosicao.TcVIS
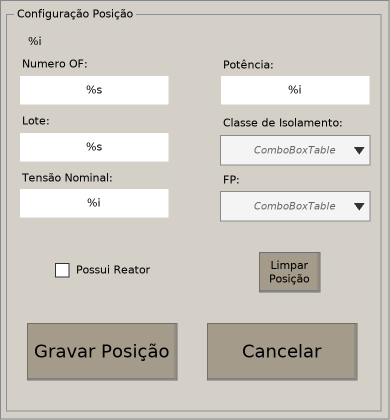
VISUALIZATION ConfigPosicao  // 390x420
VAR_IN_OUT
	bReator: BOOL;
	iOFnumber: INT;
	iSrlNumber: INT;
	
	
	
END_VAR
    GroupBox (6,6 375x405), "Configuração Posição"
        Checkbox (47,251 110x26), "Possui Reator", variable: gravarConfigPosicao.bReator[GVL.actEst]
        Button (21,317 150x57), "Gravar Posição"
            OnMouseClick: CloseDialog Dialog=ConfigPosicao, Result=OK, NumpadKeypadSet=True
            OnMouseClick: execute { gravarConfigPosicao(); }
        Button (201,317 150x57), "Cancelar"
            OnMouseClick: CloseDialog Dialog=ConfigPosicao, Result=Cancel, NumpadKeypadSet=True
        Button (253,246 61x40), "Limpar Posição"
            OnMouseClick: CloseDialog Dialog=ConfigPosicao, Result=Cancel, NumpadKeypadSet=True
            OnMouseClick: execute {
                gvl_p.aPositionsE019[gvl.actPos].numOF:='0';
                gvl_p.aPositionsE019[gvl.actPos].lote:='0';
                gvl_p.aPositionsE019[gvl.actPos].class:=0;
                gvl_p.aPositionsE019[gvl.actPos].pot:=0;
                gvl_p.aPositionsE019[gvl.actPos].cor:=0;
                IF gvl.totalPos[gvl.actEst] <> 0 THEN
                gvl.totalPos[gvl.actEst]:= gvl.totalPos[gvl.actEst] - 1;
                ELSE
                	gvl.totalPos[gvl.actEst] := 0;
                END_IF
                gravarConfigPosicao.bReator[0]:= false;
                ///// GERADOR DE LOG -------------------------------------------------------------
                gvl.envialog:= 'Posição Nº ';
                gvl.envialog:= concat(gvl.envialog, INT_TO_STRING(gvl.actPos));
                gvl.envialog:= concat(gvl.envialog,' foi limpa. ESTUFA 019');
                gvl.logRegister19:= gvl.envialog;
            }
        Label (13,43 81x30), "Numero OF:"
    Rectangle (24,30 22x23), "%i", text variable: GVL.actPos
    Textfield (19,75 150x30), "%s", text variable: GVL.cfgPos_OF019
        OnMouseDown: write the text variable via VisuDialogs.Numpad
    Label (19,163 111x30), "Tensão Nominal:"
    Textfield (220,75 150x30), "%i", text variable: GVL.cfgPos_Pot019
        OnMouseDown: write the text variable via VisuDialogs.Numpad
    Label (19,106 81x30), "Lote:"
    Label (220,165 56x30), "FP:"
    Label (220,108 144x30), "Classe de Isolamento:"
    Textfield (19,188 150x30), "%i", text variable: GVL.cfgPos_Class019
        OnMouseDown: write the text variable via VisuDialogs.Numpad
    Label (220,50 56x30), "Potência:"
    Textfield (19,132 150x30), "%s", text variable: GVL.cfgPos_LT019
        OnMouseDown: write the text variable via VisuDialogs.Keypad
    ComboBoxTable (220,135 150x30), variable: GVL.cfgPos_Iso019, data array: GVL_P.arr_Iso_1
        p3854506369: GVL_P.arr_Iso_1[INDEX]
    ComboBoxTable (220,191 150x30), variable: GVL.cfgPos_FP019, data array: GVL_P.arr_FP_1
        p3854506369: GVL_P.arr_FP_1[INDEX]
END_VISUALIZATION

// ---- VISUs/setInicio.TcVIS
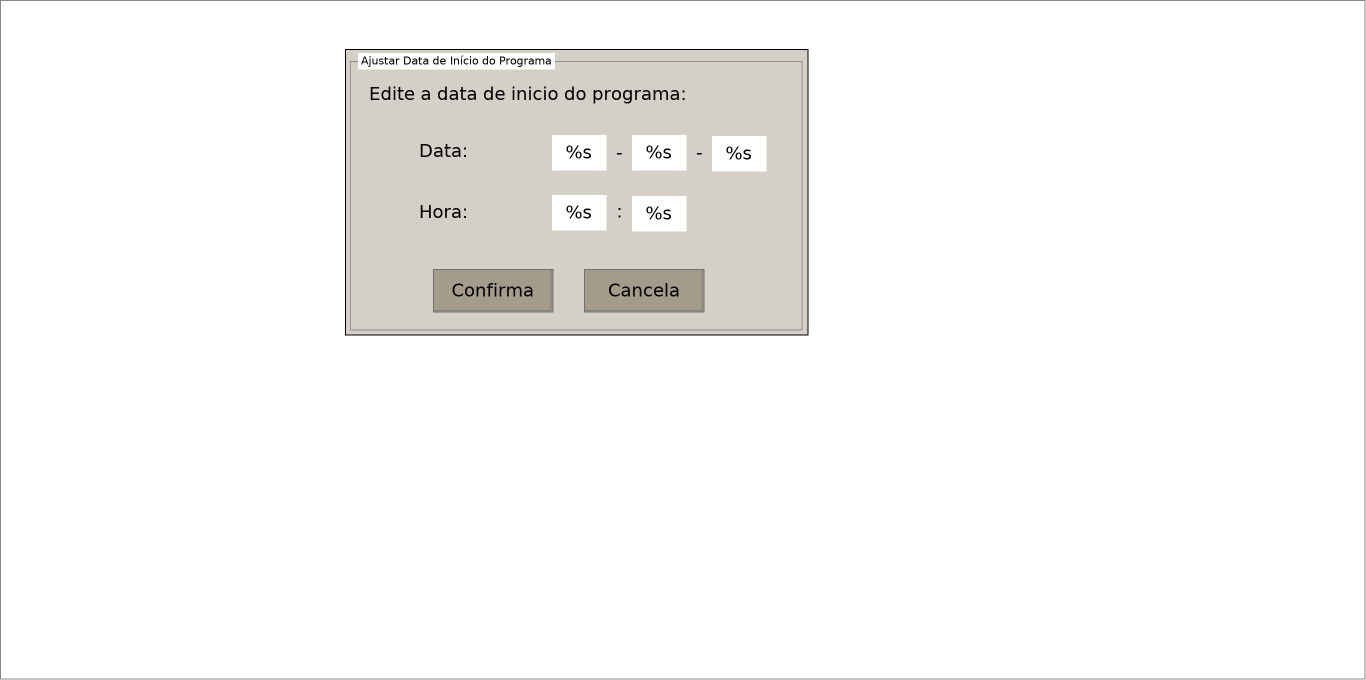
VISUALIZATION setInicio  // 1366x680
    Rectangle (345,49 463x286)
    GroupBox (350,53 452x277), "Ajustar Data de Início do Programa"
        Label (16,25 316x32), "Edite a data de inicio do programa:"
        Textfield (281,81 56x37), "%s", text variable: GVL.mes
            OnMouseClick: write the text variable via VisuDialogs.Numpad
        Textfield (361,82 56x37), "%s", text variable: GVL.ano
            OnMouseClick: write the text variable via VisuDialogs.Numpad
        Textfield (201,141 56x37), "%s", text variable: GVL.hora
            OnMouseClick: write the text variable via VisuDialogs.Numpad
        Textfield (281,142 56x37), "%s", text variable: GVL.minuto
            OnMouseClick: write the text variable via VisuDialogs.Numpad
        Label (35,144 86x30), "Hora:"
        Label (338,82 23x35), "-"
        Label (258,141 23x35), ":"
        Button (83,216 120x43), "Confirma"
            OnMouseClick: CloseDialog Dialog=setInicio, Result=OK, NumpadKeypadSet=True
            OnMouseClick: execute { confirmSetInicio(); }
        Button (234,216 120x43), "Cancela"
            OnMouseClick: CloseDialog Dialog=setInicio, Result=Cancel, NumpadKeypadSet=True
    Textfield (551,134 56x37), "%s", text variable: GVL.dia
        OnMouseClick: write the text variable via VisuDialogs.Numpad
    Label (385,136 86x30), "Data:"
    Label (608,135 23x35), "-"
END_VISUALIZATION

// ---- VISUs/setSecagem.TcVIS
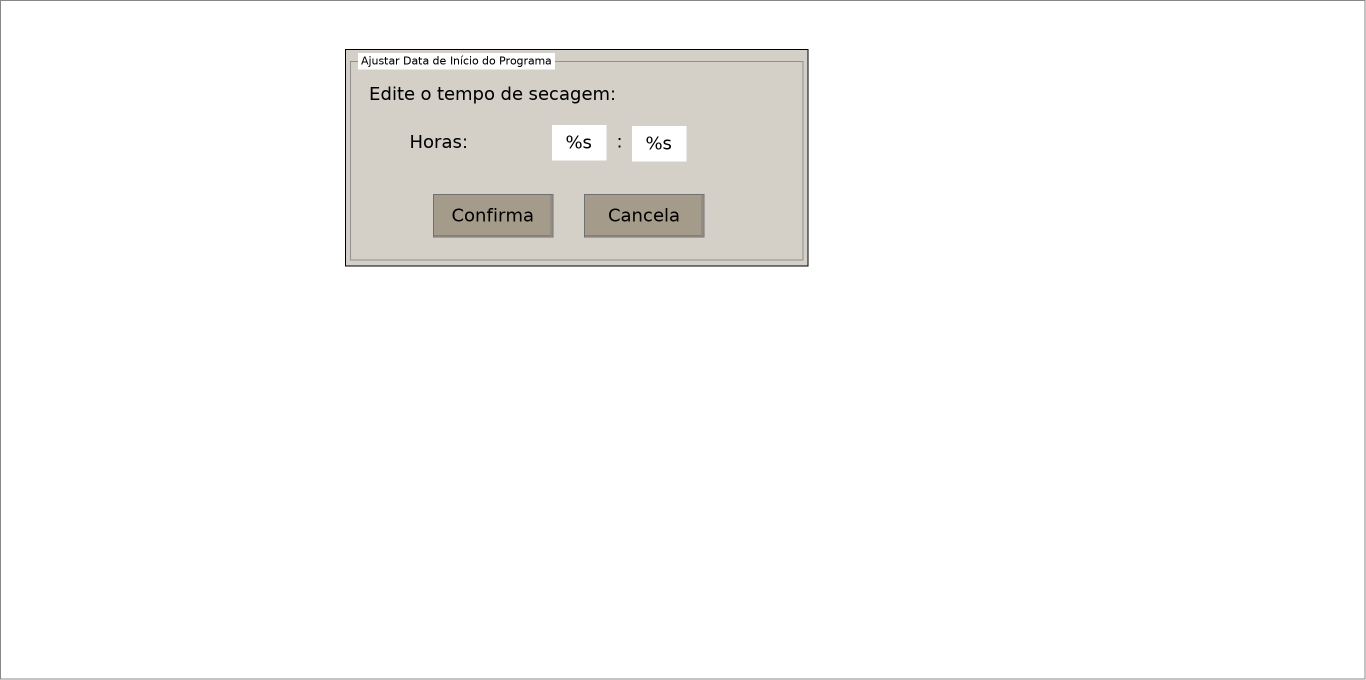
VISUALIZATION setSecagem  // 1366x680
    Rectangle (345,49 463x217)
    GroupBox (350,53 453x207), "Ajustar Data de Início do Programa"
        Label (16,25 316x32), "Edite o tempo de secagem:"
        Textfield (201,71 56x37), "%s", text variable: GVL.horaSecagem
            OnMouseClick: write the text variable via VisuDialogs.Numpad
        Textfield (281,72 56x37), "%s", text variable: GVL.minSecagem
            OnMouseClick: write the text variable via VisuDialogs.Numpad
        Label (35,74 86x30), "Horas:"
        Label (258,71 23x35), ":"
        Button (83,141 120x43), "Confirma"
            OnMouseClick: CloseDialog Dialog=setSecagem, Result=OK, NumpadKeypadSet=True
            OnMouseClick: execute { confirmSetInicio(); }
        Button (234,141 120x43), "Cancela"
            OnMouseClick: CloseDialog Dialog=setSecagem, Result=Cancel, NumpadKeypadSet=True
END_VISUALIZATION

// ---- VISUs/TimeCustom.TcVIS
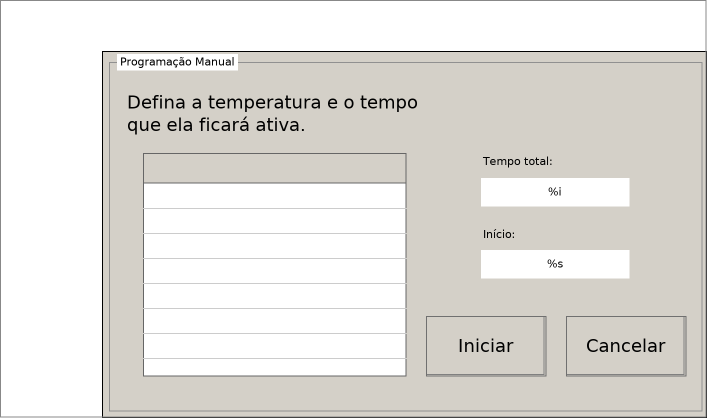
VISUALIZATION TimeCustom  // 707x418
    Rectangle (102,51 605x367)
    GroupBox (109,54 593x357), "Programação Manual"
        Button (457,262 120x60), "Cancelar"
            OnMouseClick: CloseDialog Dialog=TimeCustom, Result=OK, NumpadKeypadSet=True
        Button (317,262 120x60), "Iniciar"
            OnMouseClick: CloseDialog Dialog=TimeCustom, Result=OK, NumpadKeypadSet=True
            OnMouseClick: execute { simIniciaProg_Manual(); }
        Label (371,96 73x23), "Tempo total:"
        Textfield (371,123 150x30), "%i", text variable: GVL.totalManual[0]
    Table (143,153 263x223), data array: GVL_P.arr_CustomTime
        p3854506369: GVL_P.arr_CustomTime[0,INDEX]
        p1892666644: GVL_P.arr_CustomTime[1,INDEX]
        p2232123230: TEMPERATURA (ºC)
        p511219082: TEMPO (H)
        Columns.Column.[0].Template: OnMouseUp: write the text variable via VisuDialogs.Numpad
        Columns.Column.[1].Template: OnMouseUp: write the text variable via VisuDialogs.Numpad
    Label (124,90 305x50), "Defina a temperatura e o tempo que ela ficará ativa."
    Textfield (480,249 150x30), "%s", text variable: GVL.progInicio[GVL.actEst]
        OnMouseClick: OpenDialog Dialog=setInicio, OpenModal=True, OpenCentered=True
        OnMouseClick: execute {
            gvl.dia:= MID(STR:= gvl.progInicio[gvl.actEst] , LEN:= 2, POS:=12);
            gvl.mes:= MID(STR:= gvl.progInicio[gvl.actEst] , LEN:= 2, POS:=9);
            gvl.ano:= MID(STR:= gvl.progInicio[gvl.actEst] , LEN:= 2, POS:=6);
            gvl.hora:= MID(STR:= gvl.progInicio[gvl.actEst] , LEN:= 2, POS:=15);
            gvl.minuto:= MID(STR:= gvl.progInicio[gvl.actEst] , LEN:= 2, POS:=18);
        }
    Label (480,223 57x23), "Início:"
END_VISUALIZATION

// ---- VISUs/TimeCustom_3.TcVIS
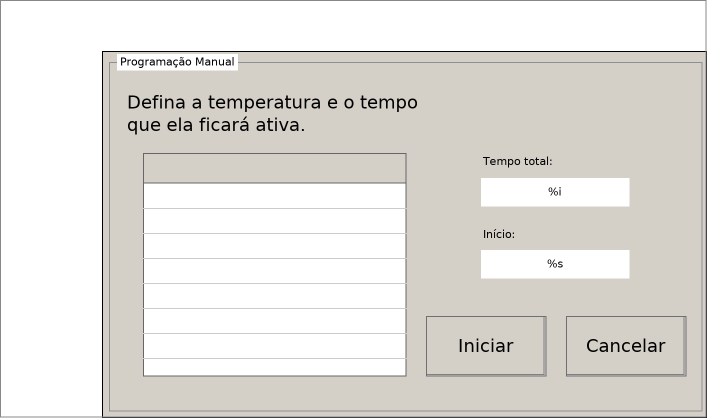
VISUALIZATION TimeCustom_3  // 707x418
    Rectangle (102,51 605x367)
    GroupBox (109,54 593x357), "Programação Manual"
        Button (457,262 120x60), "Cancelar"
            OnMouseClick: CloseDialog Dialog=TimeCustom_3, Result=OK, NumpadKeypadSet=True
        Button (317,262 120x60), "Iniciar"
            OnMouseClick: CloseDialog Dialog=TimeCustom_3, Result=OK, NumpadKeypadSet=True
            OnMouseClick: execute { simIniciaProg_Manual_3(); }
        Label (371,96 73x23), "Tempo total:"
        Textfield (371,123 150x30), "%i", text variable: GVL.totalManual[2]
    Table (143,153 263x223), data array: GVL_P.arr_CustomTime_021
        p3854506369: GVL_P.arr_CustomTime_021[0,INDEX]
        p1892666644: GVL_P.arr_CustomTime_021[1,INDEX]
        p2232123230: TEMPERATURA (ºC)
        p511219082: TEMPO (H)
        Columns.Column.[0].Template: OnMouseUp: write the text variable via VisuDialogs.Numpad
        Columns.Column.[1].Template: OnMouseUp: write the text variable via VisuDialogs.Numpad
    Label (124,90 305x50), "Defina a temperatura e o tempo que ela ficará ativa."
    Textfield (480,249 150x30), "%s", text variable: GVL.progInicio[GVL.actEst]
        OnMouseClick: OpenDialog Dialog=setInicio, OpenModal=True, OpenCentered=True
        OnMouseClick: execute {
            gvl.dia:= MID(STR:= gvl.progInicio[gvl.actEst] , LEN:= 2, POS:=12);
            gvl.mes:= MID(STR:= gvl.progInicio[gvl.actEst] , LEN:= 2, POS:=9);
            gvl.ano:= MID(STR:= gvl.progInicio[gvl.actEst] , LEN:= 2, POS:=6);
            gvl.hora:= MID(STR:= gvl.progInicio[gvl.actEst] , LEN:= 2, POS:=15);
            gvl.minuto:= MID(STR:= gvl.progInicio[gvl.actEst] , LEN:= 2, POS:=18);
        }
    Label (480,223 57x23), "Início:"
END_VISUALIZATION

// ---- VISUs/TimeCustom_2.TcVIS
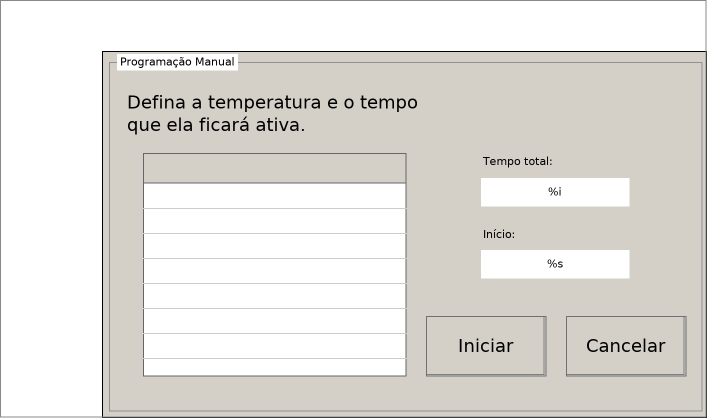
VISUALIZATION TimeCustom_2  // 707x418
    Rectangle (102,51 605x367)
    GroupBox (109,54 593x357), "Programação Manual"
        Button (457,262 120x60), "Cancelar"
            OnMouseClick: CloseDialog Dialog=TimeCustom_2, Result=OK, NumpadKeypadSet=True
        Button (317,262 120x60), "Iniciar"
            OnMouseClick: CloseDialog Dialog=TimeCustom_2, Result=OK, NumpadKeypadSet=True
            OnMouseClick: execute { simIniciaProg_Manual_2(); }
        Label (371,96 73x23), "Tempo total:"
        Textfield (371,123 150x30), "%i", text variable: GVL.totalManual[1]
    Table (143,153 263x223), data array: GVL_P.arr_CustomTime_020
        p3854506369: GVL_P.arr_CustomTime_020[0,INDEX]
        p1892666644: GVL_P.arr_CustomTime_020[1,INDEX]
        p2232123230: TEMPERATURA (ºC)
        p511219082: TEMPO (H)
        Columns.Column.[0].Template: OnMouseUp: write the text variable via VisuDialogs.Numpad
        Columns.Column.[1].Template: OnMouseUp: write the text variable via VisuDialogs.Numpad
    Label (124,90 305x50), "Defina a temperatura e o tempo que ela ficará ativa."
    Textfield (480,249 150x30), "%s", text variable: GVL.progInicio[GVL.actEst]
        OnMouseClick: OpenDialog Dialog=setInicio, OpenModal=True, OpenCentered=True
        OnMouseClick: execute {
            gvl.dia:= MID(STR:= gvl.progInicio[gvl.actEst] , LEN:= 2, POS:=12);
            gvl.mes:= MID(STR:= gvl.progInicio[gvl.actEst] , LEN:= 2, POS:=9);
            gvl.ano:= MID(STR:= gvl.progInicio[gvl.actEst] , LEN:= 2, POS:=6);
            gvl.hora:= MID(STR:= gvl.progInicio[gvl.actEst] , LEN:= 2, POS:=15);
            gvl.minuto:= MID(STR:= gvl.progInicio[gvl.actEst] , LEN:= 2, POS:=18);
        }
    Label (480,223 57x23), "Início:"
END_VISUALIZATION
